// POUs/BACnet Objects/Local (Server)/Extended Process Data/FB_BACnet_PulseConverter_EX
FUNCTION_BLOCK FB_BACnet_PulseConverter_EX
VAR_IN_OUT
	Device				: FB_BACnet_Device;
END_VAR
VAR_OUTPUT
	bReady				: BOOL;
	fPresentValue		: REAL;
	bHighLimitEn		: BOOL;
	fHighLimit			: REAL;
	bLowLimitEn			: BOOL;
	fLowLimit			: REAL;
	fAdjustValue		: REAL;
	nCount				: UDINT;
	nCountBeforeChg		: UDINT;
	bOverridden			: BOOL;
	bOutOfService		: BOOL;
	bFault				: BOOL;
	bInAlarm			: BOOL;
	bOverRange			: BOOL;
	bUnderRange			: BOOL;
	bNoSensor			: BOOL;
	bOpenLoop			: BOOL;
	bShortedLoop		: BOOL;
	bCommFailure		: BOOL;
	bConfigError		: BOOL;
	bOtherFault			: BOOL;
	eEventState			: E_BACNETEVENTSTATE;
	bAckedTrans_ToOffNormal : BOOL;
	bAckedTrans_ToFault		: BOOL;
	bAckedTrans_ToNormal	: BOOL;
	tObjectID			: T_BACnet_ObjectIdentifier := 16#FFFFFFFF;
	bError				: BOOL;
	nErrorId			: UINT;
END_VAR
VAR
	_PresentValueIn AT%I*: REAL; 	(* ~(BACnet_PresentValue 		:		: )
								   		(BACnet_ObjectType 			: PC	: )	*)
	_HighLimit AT%I*: REAL;			(* ~(BACnet_HighLimit			:		: )	*)
	_LowLimit AT%I*: REAL;			(* ~(BACnet_LowLimit			:		: )	*)
	_AdjustValue AT%I*: REAL;		(* ~(BACnet_AdjustValue 		:		: ) *)
	_Count AT%I*: UDINT;			(* ~(BACnet_Count		 		:		: ) *)
	_CountBeforeChange AT%I*: UDINT;(* ~(BACnet_CountBeforeChange	:		: ) *)
	_ObjectId AT%I* : DWORD;		(* ~(BACnet_ObjectIdentifier	:		: LINK) *)
	_StatusFlags AT%I*: WORD; 		(* ~(BACnet_StatusFlags 		:		: )	*)
	_AckedTransitions AT%I*:WORD;	(* ~(BACnet_AckedTransitions	:		: ) *)
	_EventState AT%I*: WORD; 		(* ~(BACnet_EventState			:		: )	*)
	_LimitEnable AT%I*: WORD;		(* ~(BACnet_LimitEnable			:		: )	*)
	_Reliability AT%I*: WORD;;		(* ~(BACnet_Reliability 		:		: )	*)
	_AckedTransBits : ST_BACnet_EventTransitionBits;
	_StatusFlagsBits : ST_BACnet_StatusFlags;
	_LimitEnableBits : ST_BACnet_LimitEnable;
	_nUpdateCount : UDINT := 0;
END_VAR

(* update server device *)
IF (Device._nUpdateCount = _nUpdateCount) THEN
	Device();
END_IF
(* remind current number of update counter *)
_nUpdateCount := Device._nUpdateCount;

IF Device.bFirstCycle THEN
	(* first call of the server device since reboot/reset *)
	bReady := FALSE;

ELSIF (F_BACnet_GetObjType(_ObjectId) <> BACnetObjectType_PulseConverter) THEN
	(* wrong mapping / invalid object ID *)
	IF _ObjectId = 0 THEN
		nErrorId := BACnet_ERR_WRONG_MAPPING;
	ELSE
		nErrorId := BACnet_ERR_INVALID_OBJECTID;
	END_IF
	bReady := FALSE;
	tObjectID := 16#FFFFFFFF;

ELSIF (_StatusFlags < 4) THEN
	(* wrong mapping *)
	nErrorId := BACnet_ERR_WRONG_MAPPING;
	bReady := FALSE;

ELSIF Device.bOperational THEN
	(* ready state *)
	bReady := TRUE;
	nErrorId := BACnet_ERR_NO_ERROR;

	(* present value *)
	fPresentValue := _PresentValueIn;

	(* build bit states *)
	_StatusFlagsBits := F_BACnet_StatusFlags(_StatusFlags);
	_AckedTransBits := F_BACnet_EventTransitionFlags(_AckedTransitions);
	_LimitEnableBits :=	F_BACnet_LimitEnableFlags(_LimitEnable);

	(* copy states to output *)
	bHighLimitEn:= _LimitEnableBits.highLimitEnable;
	bLowLimitEn	:= _LimitEnableBits.lowLimitEnable;
	bOverridden	:= _StatusFlagsBits.overridden;
	bOutOfService:= _StatusFlagsBits.out_of_service;
	bFault		:= _StatusFlagsBits.fault;
	bInAlarm	:= _StatusFlagsBits.in_alarm;
	bOverRange	:= (_Reliability = TO_WORD(BACnetReliability_over_range));
	bUnderRange	:= (_Reliability = TO_WORD(BACnetReliability_under_range));
	bNoSensor	:= (_Reliability = TO_WORD(BACnetReliability_no_sensor));
	bOpenLoop	:= (_Reliability = TO_WORD(BACnetReliability_open_loop));
	bShortedLoop:= (_Reliability = TO_WORD(BACnetReliability_shorted_loop));
	bCommFailure := (_Reliability = TO_WORD(BACnetReliability_communication_failure));
	bConfigError:= (_Reliability = TO_WORD(BACnetReliability_configuration_error));
	bOtherFault	:= (_Reliability = TO_WORD(BACnetReliability_unreliable_other));
	bAckedTrans_ToOffNormal := _AckedTransBits.to_offnormal;
	bAckedTrans_ToFault := _AckedTransBits.to_fault;
	bAckedTrans_ToNormal := _AckedTransBits.to_normal;

	(* convert enumeration *)
	eEventState := TO_INT(_EventState);

	(* additional information *)
	fHighLimit			:= _HighLimit;
	fLowLimit			:= _LowLimit;
	fAdjustValue		:= _AdjustValue;
	nCount				:= _Count;
	nCountBeforeChg		:= _CountBeforeChange;
	tObjectID		:= F_BACnet_GetObjInstance(_ObjectId);

ELSE
	(* server device not ready, reset local ready flag *)
	bReady := FALSE;
	nErrorId := BACnet_ERR_OPERATIONAL;
END_IF
(* set error flag *)
bError := (nErrorId <> BACnet_ERR_NO_ERROR);

END_FUNCTION_BLOCK

// POUs/BACnet Objects/Local (Server)/Extended Process Data/FB_BACnet_Schedule_EX
FUNCTION_BLOCK FB_BACnet_Schedule_EX
VAR_IN_OUT
	Device				: FB_BACnet_Device;
END_VAR
VAR_OUTPUT
	bReady				: BOOL;
	bPresentValue		: BOOL;
	bOverridden			: BOOL;
	bOutOfService		: BOOL;
	bFault				: BOOL;
	bInAlarm			: BOOL;
	bConfigError		: BOOL;
	bOtherFault			: BOOL;
	tObjectID			: T_BACnet_ObjectIdentifier := 16#FFFFFFFF;
	bError				: BOOL;
	nErrorId			: UINT;
END_VAR
VAR
	_ObjectId AT%I*: DWORD;		(* ~(BACnet_ObjectIdentifier		:		: LINK) *)
	_Reliability AT%I*: WORD;; 	(* ~(BACnet_Reliability 			:		: )	*)
	_StatusFlags AT%I*: WORD; 	(* ~(BACnet_StatusFlags 			:		: )	*)
	_PresentValue AT%I*: BOOL;	(* ~(BACnet_PresentValueBool 		:		: )
									(BACnet_ObjectType 				: SCHED	: )	*)
	_StatusFlagsBits : ST_BACnet_StatusFlags;
	_nUpdateCount : UDINT := 0;
END_VAR

(* update server device *)
IF (Device._nUpdateCount = _nUpdateCount) THEN
	Device();
END_IF
(* remind current number of update counter *)
_nUpdateCount := Device._nUpdateCount;

(* check object type *)
IF (F_BACnet_GetObjType(_ObjectId) <> BACnetObjectType_Schedule) THEN
	(* wrong mapping / invalid object ID *)
	IF _ObjectId = 0 THEN
		nErrorId := BACnet_ERR_WRONG_MAPPING;
	ELSE
		nErrorId := BACnet_ERR_INVALID_OBJECTID;
	END_IF
	bReady := FALSE;

ELSIF (_StatusFlags < 4) THEN
	(* wrong mapping *)
	nErrorId := BACnet_ERR_WRONG_MAPPING;
	bReady := FALSE;

ELSIF Device.bOperational THEN
	(* ready state *)
	bReady := TRUE;
	nErrorId := BACnet_ERR_NO_ERROR;

	(* present value *)
	bPresentValue := _PresentValue;

	(* build bit states *)
	_StatusFlagsBits := F_BACnet_StatusFlags(_StatusFlags);

	(* copy states to output *)
	bOverridden := _StatusFlagsBits.overridden;
	bOutOfService := _StatusFlagsBits.out_of_service;
	bFault := _StatusFlagsBits.fault;
	bInAlarm := _StatusFlagsBits.in_alarm;
	bConfigError := (_Reliability = TO_WORD(BACnetReliability_configuration_error));
	bOtherFault := (_Reliability = TO_WORD(BACnetReliability_unreliable_other));
	tObjectID := _ObjectId;

ELSE
	bReady := FALSE;
	nErrorId := BACnet_ERR_OPERATIONAL;
END_IF
(* set error flag *)
bError := (nErrorId <> BACnet_ERR_NO_ERROR);

END_FUNCTION_BLOCK

// POUs/BACnet Objects/Local (Server)/Extended Process Data/FB_BACnet_TrendLog_EX
FUNCTION_BLOCK FB_BACnet_TrendLog_EX
VAR_IN_OUT
	Device	: FB_BACnet_Device;
END_VAR
VAR_OUTPUT
	bReady			: BOOL;
	bLogEnable		: BOOL;
	nRecordCount	: UDINT;
	nTotalCount		: UDINT;
	eEventState		: E_BACNETEVENTSTATE;
	bAckedTrans_ToOffNormal : BOOL;
	bAckedTrans_ToFault		: BOOL;
	bAckedTrans_ToNormal	: BOOL;
	tObjectID		: T_BACnet_ObjectIdentifier := 16#FFFFFFFF;
	bError			: BOOL;
	nErrorId		: UINT;
END_VAR
VAR
	_RecordCount AT%I*: UDINT;		(* ~(BACnet_RecordCount			:		: )
										(BACnet_ObjectType			: TLOG	: )	*)
	_TotalRecordCount AT%I*: UDINT;	(* ~(BACnet_TotalRecordCount	:		: )	*)
	_ObjectId AT%I*: DWORD;			(* ~(BACnet_ObjectIdentifier	:		: LINK) *)
	_EventState AT%I*: WORD;		(* ~(BACnet_EventState			:		: )	*)
	_AckedTransitions AT%I*:WORD;	(* ~(BACnet_AckedTransitions	:		: ) *)
	_LogEnable AT%I*: BOOL;			(* ~(BACnet_LogEnable			: 		: )	*)
	_AckedTransBits : ST_BACnet_EventTransitionBits;
	_nUpdateCount : UDINT := 0;
END_VAR

(* update server device *)
IF (Device._nUpdateCount = _nUpdateCount) THEN
	Device();
END_IF
(* remind current number of update counter *)
_nUpdateCount := Device._nUpdateCount;

(* check object type *)
IF (F_BACnet_GetObjType(_ObjectId) <> BACnetObjectType_TrendLog) THEN
	(* wrong mapping / invalid object ID *)
	IF _ObjectId = 0 THEN
		nErrorId := BACnet_ERR_WRONG_MAPPING;
	ELSE
		nErrorId := BACnet_ERR_INVALID_OBJECTID;
	END_IF
	bReady := FALSE;

ELSIF Device.bOperational THEN
	(* ready state *)
	bReady := TRUE;
	bLogEnable := _LogEnable;
	nErrorId := BACnet_ERR_NO_ERROR;

	(* build bit states *)
	_AckedTransBits		:= F_BACnet_EventTransitionFlags(_AckedTransitions);
	bAckedTrans_ToOffNormal := _AckedTransBits.to_offnormal;
	bAckedTrans_ToFault := _AckedTransBits.to_fault;
	bAckedTrans_ToNormal := _AckedTransBits.to_normal;
	tObjectID := _ObjectId;

	(* convert enumeration *)
	eEventState := TO_INT(_EventState);

	(* other states *)
	nRecordCount := _RecordCount;
	nTotalCount := _TotalRecordCount;

ELSE
	bReady := FALSE;
	nErrorId := BACnet_ERR_OPERATIONAL;
END_IF
(* set error flag *)
bError := (nErrorId <> BACnet_ERR_NO_ERROR);

END_FUNCTION_BLOCK

// POUs/BACnet Objects/Local (Server)/R6/FB_BACnet_Accumulator_R6
FUNCTION_BLOCK FB_BACnet_Accumulator_R6
VAR_INPUT
	nPV					: UDINT; (* number for present_value *)
END_VAR
VAR_IN_OUT
	Device				: FB_BACnet_Device;
END_VAR
VAR_OUTPUT
	bReady				: BOOL;
	nPresentValue		: UDINT;
	bOverridden			: BOOL;
	bOutOfService		: BOOL;
	bFault				: BOOL;
	bInAlarm			: BOOL;
	bError				: BOOL;
	nErrorId			: UINT;
END_VAR
VAR
	_PresentValueIn AT%I*:UDINT;	(* ~(BACnet_PresentValue	:		: )
										(BACnet_MaxPresValue	:		: writeprotect,nolink)
										(BACnet_ObjectType		: ACC	: )	*)
    _PresentValueOut AT%Q*:UDINT;	(* ~(BACnet_PresentValue	:		: )	*)
	_StatusFlags AT%I*:WORD;		(* ~(BACnet_StatusFlags		:		: )	*)
	_StatusFlagsBits : ST_BACnet_StatusFlags;

	_nUpdateCount : UDINT := 0;
END_VAR

(* update device *)
IF (Device._nUpdateCount = _nUpdateCount) THEN
	Device();
END_IF
(* remind current number of update counter *)
_nUpdateCount := Device._nUpdateCount;

IF _StatusFlags < 4 THEN
	(* mapping seems to be wrong (bit string for status flags must be 4 in minimum) *)
	nErrorId := BACnet_ERR_WRONG_MAPPING;

ELSIF Device.bOperational THEN
	(* clear error flag *)
	nErrorId := BACnet_ERR_NO_ERROR;
	bReady := TRUE;
	(* copy present value *)
	nPresentValue 		:= _PresentValueIn;
	_PresentValueOut	:= nPV;

	(* build bit states *)
	_StatusFlagsBits	:= F_BACnet_StatusFlags(_StatusFlags);

	(* copy states to output *)
	bOverridden := _StatusFlagsBits.overridden;
	bOutOfService := _StatusFlagsBits.out_of_service;
	bFault := _StatusFlagsBits.fault;
	bInAlarm := _StatusFlagsBits.in_alarm;
ELSE
	bReady := FALSE;
	(* and set error ID *)
	nErrorId := BACnet_ERR_OPERATIONAL;
END_IF

(* set error flag *)
bError := (nErrorId <> BACnet_ERR_NO_ERROR);

END_FUNCTION_BLOCK

// POUs/BACnet Objects/Local (Server)/R6/FB_BACnet_Accumulator_RAW_R6
FUNCTION_BLOCK FB_BACnet_Accumulator_RAW_R6
VAR_INPUT
	nPV					: UDINT; (* number for present_value *)
	nReliability		: WORD;
	bOutOfServiceOut	: BOOL;
END_VAR
VAR_IN_OUT
	Device				: FB_BACnet_Device;
END_VAR
VAR_OUTPUT
	bReady				: BOOL;
	nPresentValue		: UDINT;
	nMaxPV				: UDINT;
	bOverridden			: BOOL;
	bOutOfService		: BOOL;
	bFault				: BOOL;
	bInAlarm			: BOOL;
	bOverRange			: BOOL;
	bUnderRange			: BOOL;
	bNoSensor			: BOOL;
	bOpenLoop			: BOOL;
	bShortedLoop		: BOOL;
	bOtherFault			: BOOL;
	eEventState			: E_BACNETEVENTSTATE;
	bError				: BOOL;
	nErrorId			: UINT;
END_VAR
VAR
	_PresentValueIn AT%I*:UDINT;	(* ~(BACnet_PresentValue	:		: )
										(BACnet_ObjectType		: ACC	: )	*)
    _PresentValueOut AT%Q*:UDINT;	(* ~(BACnet_PresentValue	:		: )	*)
	_MaxPresValue AT%I*:UDINT;		(* ~(BACnet_MaxPresValue	:		: writeprotect) *)
	_StatusFlags AT%I*:WORD;		(* ~(BACnet_StatusFlags		:		: )	*)
	_EventState AT%I*: WORD; 		(* ~(BACnet_EventState 		:		: )	*)
	_Reliability AT%I*: WORD;; 		(* ~(BACnet_Reliability 	:		: )	*)
	_StatusFlagsOut AT%Q*:WORD;		(* ~(BACnet_StatusFlags		:		: )	*)
	_EventStateOut AT%Q*: WORD;		(* ~(BACnet_EventState 		:		: )	*)
	_ReliabilityOut AT%Q*: WORD;	(* ~(BACnet_Reliability 	:		: )	*)
	_OutOfServiceOut AT%Q*: BOOL;	(* ~(BACnet_OutOfService	:		: writeprotect) *)
	_StatusFlagsBits : ST_BACnet_StatusFlags;
	_StatusFlagsOutBits : ST_BACnet_StatusFlags;
	_nUpdateCount : UDINT := 0;
END_VAR

(* update client device *)
IF (Device._nUpdateCount = _nUpdateCount) THEN
	Device();
END_IF
(* remind current number of update counter *)
_nUpdateCount := Device._nUpdateCount;

(* copy reliability and out of service flags *)
_ReliabilityOut		:= nReliability;
_OutOfServiceOut	:= bOutOfServiceOut;

IF _StatusFlags < 4 THEN
	(* mapping seems to be wrong (bit string for status flags must be 4 in minimum) *)
	nErrorId := BACnet_ERR_WRONG_MAPPING;

ELSIF Device.bOperational THEN
	(* clear error flag *)
	nErrorId := BACnet_ERR_NO_ERROR;
	bReady := TRUE;
	(* copy present value *)
	nPresentValue 		:= _PresentValueIn;
	_PresentValueOut	:= nPV;
	nMaxPV				:= _MaxPresValue;

	(* build bit states *)
	_StatusFlagsBits	:= F_BACnet_StatusFlags(_StatusFlags);

	(* copy states to output *)
	bOverridden := _StatusFlagsBits.overridden;
	bOutOfService := _StatusFlagsBits.out_of_service;
	bFault := _StatusFlagsBits.fault;
	bInAlarm := _StatusFlagsBits.in_alarm;
	bOverRange := (_Reliability = TO_WORD(BACnetReliability_over_range));
	bUnderRange := (_Reliability = TO_WORD(BACnetReliability_under_range));
	bNoSensor := (_Reliability = TO_WORD(BACnetReliability_no_sensor));
	bOpenLoop := (_Reliability = TO_WORD(BACnetReliability_open_loop));
	bShortedLoop := (_Reliability = TO_WORD(BACnetReliability_shorted_loop));
	bOtherFault := (_Reliability = TO_WORD(BACnetReliability_unreliable_other));

	(* convert enumeration *)
	eEventState := TO_INT(_EventState);
ELSE
	bReady := FALSE;
	(* and set error ID *)
	nErrorId := BACnet_ERR_OPERATIONAL;
END_IF

(* set status flags depending on reliability *)
IF TO_INT(_ReliabilityOut) = BACnetReliability_no_fault_detected THEN
	_StatusFlagsOutBits.fault := FALSE;
	_StatusFlagsOutBits.in_alarm := FALSE;
	_EventStateOut := 0;
ELSE
	_StatusFlagsOutBits.fault := TRUE;
	_StatusFlagsOutBits.in_alarm := TRUE;
	_EventStateOut := 1;
END_IF

_StatusFlagsOutBits.out_of_service := _OutOfServiceOut;
_StatusFlagsOut	:= F_BACnet_GetStatusFlagsData(_StatusFlagsOutBits);

(* set error flag *)
bError := (nErrorId <> BACnet_ERR_NO_ERROR);

END_FUNCTION_BLOCK

// POUs/BACnet Objects/Local (Server)/RAW/FB_BACnet_Accumulator_RAW
FUNCTION_BLOCK FB_BACnet_Accumulator_RAW
VAR_INPUT
	nRawIn				AT%Q*: UINT; (* ~(BACnet_RawIoAccumulatorUnsignedValue : : ) *)
	bNoSensor			: BOOL;
	bOverRange			: BOOL;
	bUnderRange			: BOOL;
	bOpenLoop			: BOOL;
	bShortedLoop		: BOOL;
	bCommFailure		: BOOL;
	bOtherFault			: BOOL;
END_VAR
VAR_IN_OUT
	Device				: FB_BACnet_Device;
END_VAR
VAR_OUTPUT
	bReady				: BOOL;
	nPresentValue		: UDINT;
	bOverridden			: BOOL;
	bOutOfService		: BOOL;
	bFault				: BOOL;
	bInAlarm			: BOOL;
	bError				: BOOL;
	nErrorId			: UINT;
END_VAR
VAR
	_PresentValueIn AT%I*:UDINT;	(* ~(BACnet_PresentValue	:		: )
										(BACnet_MaxPresValue	:		: writeprotect,nolink)
										(BACnet_ObjectType		: ACC	: )	*)
	_ObjectId AT%I*: DWORD;			(* ~(BACnet_ObjectIdentifier:		: LINK) *)
	_StatusFlags AT%I*:WORD;		(* ~(BACnet_StatusFlags		:		: )	*)
	_ReliabilityIn AT%I*: WORD;		(* ~(BACnet_Reliability 	:		: )	*)
	_ReliabilityOut AT%Q*: WORD := INT_TO_WORD(BACnetReliability_no_fault_detected);(* ~(BACnet_Reliability 	:		: )	*)
	_StatusFlagsBits : ST_BACnet_StatusFlags;

	_nUpdateCount : UDINT := 0;
END_VAR

(* update device *)
IF Device._nUpdateCount = _nUpdateCount THEN
	Device();
END_IF
(* remind current number of update counter *)
_nUpdateCount := Device._nUpdateCount;

(* handle raw error *)
IF bNoSensor THEN
	_ReliabilityOut := TO_WORD(BACnetReliability_no_sensor);
ELSIF bOverRange THEN
	_ReliabilityOut := TO_WORD(BACnetReliability_over_range);
ELSIF bUnderRange THEN
	_ReliabilityOut := TO_WORD(BACnetReliability_under_range);
ELSIF bOpenLoop THEN
	_ReliabilityOut := TO_WORD(BACnetReliability_open_loop);
ELSIF bShortedLoop THEN
	_ReliabilityOut := TO_WORD(BACnetReliability_shorted_loop);
ELSIF bCommFailure THEN
	_ReliabilityOut := TO_WORD(BACnetReliability_communication_failure);
ELSIF bOtherFault THEN
	_ReliabilityOut := TO_WORD(BACnetReliability_unreliable_other);
ELSE
	_ReliabilityOut := TO_WORD(BACnetReliability_no_fault_detected);
END_IF

IF _StatusFlags < 4 THEN
	(* mapping seems to be wrong (bit string for status flags must be 4 in minimum) *)
	nErrorId := BACnet_ERR_WRONG_MAPPING;

ELSIF Device.bOperational THEN
	(* clear error flag *)
	nErrorId := BACnet_ERR_NO_ERROR;
	bReady := TRUE;
	(* copy present value *)
	nPresentValue 		:= _PresentValueIn;

	(* build bit states *)
	_StatusFlagsBits	:= F_BACnet_StatusFlags(_StatusFlags);

	(* copy states to output *)
	bOverridden := _StatusFlagsBits.overridden;
	bOutOfService := _StatusFlagsBits.out_of_service;
	bFault := _StatusFlagsBits.fault;
	bInAlarm := _StatusFlagsBits.in_alarm;
ELSE
	bReady := FALSE;
	(* and set error ID *)
	nErrorId := BACnet_ERR_OPERATIONAL;
END_IF

(* set error flag *)
bError := (nErrorId <> BACnet_ERR_NO_ERROR);

END_FUNCTION_BLOCK

// POUs/BACnet Objects/Local (Server)/RAW/FB_BACnet_AnalogInput_RAW
FUNCTION_BLOCK FB_BACnet_AnalogInput_RAW
VAR_INPUT
	nRawIn			AT%Q*: INT; (* ~(BACnet_RawIoAnalogSignedValue : : ) *)
	bNoSensor		: BOOL;
	bOverRange		: BOOL;
	bUnderRange		: BOOL;
	bOpenLoop		: BOOL;
	bShortedLoop	: BOOL;
	bCommFailure	: BOOL;
	bOtherFault		: BOOL;
END_VAR
VAR_IN_OUT
	Device	: FB_BACnet_Device;
END_VAR
VAR_OUTPUT
	bReady			: BOOL;
	fPresentValue	: REAL;
	bOverridden		: BOOL;
	bOutOfService	: BOOL;
	bFault			: BOOL;
	bInAlarm		: BOOL;
	bAckedTrans_ToOffNormal : BOOL;
	bAckedTrans_ToFault		: BOOL;
	bAckedTrans_ToNormal	: BOOL;
	bError			: BOOL;
	nErrorId		: UINT;
END_VAR
VAR
	_Reliability AT%Q*: WORD := INT_TO_WORD(BACnetReliability_no_fault_detected);(* ~(BACnet_Reliability 	:		: )	*)
	_PresentValue AT%I*: REAL; 		(* ~(BACnet_PresentValue 	:		: )
								   		(BACnet_ObjectType 		: AI	: )	*)
	_ObjectId AT%I*: DWORD;			(* ~(BACnet_ObjectIdentifier:		: LINK) *)
	_AckedTransitions AT%I*:WORD;	(* ~(BACnet_AckedTransitions:		: ) *)
	_StatusFlags AT%I*: WORD; 		(* ~(BACnet_StatusFlags 	:		: )	*)
	_AckedTransBits : ST_BACnet_EventTransitionBits;
	_StatusFlagsBits : ST_BACnet_StatusFlags;
	_nUpdateCount : UDINT := 0;
END_VAR

(* update server device *)
IF (Device._nUpdateCount = _nUpdateCount) THEN
	Device();
END_IF
(* remind current number of update counter *)
_nUpdateCount := Device._nUpdateCount;

(* handle raw error *)
IF bNoSensor THEN
	_Reliability := TO_WORD(BACnetReliability_no_sensor);
ELSIF bOverRange THEN
	_Reliability := TO_WORD(BACnetReliability_over_range);
ELSIF bUnderRange THEN
	_Reliability := TO_WORD(BACnetReliability_under_range);
ELSIF bOpenLoop THEN
	_Reliability := TO_WORD(BACnetReliability_open_loop);
ELSIF bShortedLoop THEN
	_Reliability := TO_WORD(BACnetReliability_shorted_loop);
ELSIF bCommFailure THEN
	_Reliability := TO_WORD(BACnetReliability_communication_failure);
ELSIF bOtherFault THEN
	_Reliability := TO_WORD(BACnetReliability_unreliable_other);
ELSE
	_Reliability := TO_WORD(BACnetReliability_no_fault_detected);
END_IF

(* check BitString format of StatusFlags --> if StatusFlags are less than 4, object isn't linked correctly *)
IF (_StatusFlags < 4) THEN
	(* wrong mapping *)
	nErrorId := BACnet_ERR_WRONG_MAPPING;
	bReady := FALSE;

ELSIF Device.bOperational THEN
	(* ready state *)
	bReady := TRUE;
	nErrorId := BACnet_ERR_NO_ERROR;

	(* present value *)
	fPresentValue := _PresentValue;

	(* build bit states *)
	_StatusFlagsBits := F_BACnet_StatusFlags(_StatusFlags);
	_AckedTransBits		:= F_BACnet_EventTransitionFlags(_AckedTransitions);

	(* copy states to output *)
	bOverridden := _StatusFlagsBits.overridden;
	bOutOfService := _StatusFlagsBits.out_of_service;
	bFault := _StatusFlagsBits.fault;
	bInAlarm := _StatusFlagsBits.in_alarm;
	bAckedTrans_ToOffNormal := _AckedTransBits.to_offnormal;
	bAckedTrans_ToFault := _AckedTransBits.to_fault;
	bAckedTrans_ToNormal := _AckedTransBits.to_normal;
ELSE
	(* server device not ready, reset local ready also *)
	bReady := FALSE;
	nErrorId := BACnet_ERR_OPERATIONAL;
END_IF
(* set error flag *)
bError := (nErrorId <> BACnet_ERR_NO_ERROR);

END_FUNCTION_BLOCK

// POUs/BACnet Objects/Local (Server)/RAW/FB_BACnet_AnalogOutput_RAW
FUNCTION_BLOCK FB_BACnet_AnalogOutput_RAW
VAR_INPUT
	bEnablePV		: BOOL; (* enable present value with priority x in priority array, FALSE = priority x disable *)
	bNullPV			: BOOL; (* clear priority entry *)
	fPV				: REAL; (* decimal number for priority x, when input bEnablePV is TRUE *)
	bRawOverridden	AT%Q*: BOOL; (* ~(BACnet_RawIoStateOverride	:		: ) *)
	bNoOutput		: BOOL;
	bOpenLoop		: BOOL;
	bShortedLoop	: BOOL;
	bCommFailure	: BOOL;
	bOtherFault		: BOOL;
END_VAR
VAR_IN_OUT
	Device	: FB_BACnet_Device;
END_VAR
VAR_OUTPUT
	bReady			: BOOL;
	fPresentValue	: REAL;
	bOverridden		: BOOL;
	bOutOfService	: BOOL;
	bFault			: BOOL;
	bInAlarm		: BOOL;
	bAckedTrans_ToOffNormal : BOOL;
	bAckedTrans_ToFault		: BOOL;
	bAckedTrans_ToNormal	: BOOL;
	bError			: BOOL;
	nErrorId		: UINT;
	nRawOut			AT%I*: INT;			(* ~(BACnet_RawIoAnalogSignedValue : : ) *)
END_VAR
VAR
	_PresentValue AT%I*: REAL; 			(* ~(BACnet_PresentValue 			:		: )
								   			(BACnet_ObjectType 				: AO	: )	*)
	_ObjectId AT%I*: DWORD;				(* ~(BACnet_ObjectIdentifier		:		: LINK) *)
	_AckedTransitions AT%I*:WORD;		(* ~(BACnet_AckedTransitions		:		: ) *)
	_StatusFlags AT%I*: WORD; 			(* ~(BACnet_StatusFlags 			:		: )	*)
    _PresentValue_Priority12 AT%Q*: DWORD;(* ~(BACnet_PresentValue_Priority12:		: )	*)
	_Reliability AT%Q*: WORD := INT_TO_WORD(BACnetReliability_no_fault_detected);(* ~(BACnet_Reliability 	:		: )	*)
	_AckedTransBits : ST_BACnet_EventTransitionBits;
	_StatusFlagsBits : ST_BACnet_StatusFlags;
	_nUpdateCount : UDINT := 0;
END_VAR

(* update server device *)
IF (Device._nUpdateCount = _nUpdateCount) THEN
	Device();
END_IF
(* remind current number of update counter *)
_nUpdateCount := Device._nUpdateCount;

(* handle raw error *)
IF bNoOutput THEN
	_Reliability := TO_WORD(BACnetReliability_no_output);
ELSIF bOpenLoop THEN
	_Reliability := TO_WORD(BACnetReliability_open_loop);
ELSIF bShortedLoop THEN
	_Reliability := TO_WORD(BACnetReliability_shorted_loop);
ELSIF bCommFailure THEN
	_Reliability := TO_WORD(BACnetReliability_communication_failure);
ELSIF bOtherFault THEN
	_Reliability := TO_WORD(BACnetReliability_unreliable_other);
ELSE
	_Reliability := TO_WORD(BACnetReliability_no_fault_detected);
END_IF

IF Device.bFirstCycle THEN
	(* first call of the server device since reboot/reset *)
	bReady := FALSE;
	_PresentValue_Priority12 := F_BACnet_RealNothing();

ELSIF (_StatusFlags < 4) THEN
	(* wrong mapping *)
	nErrorId := BACnet_ERR_WRONG_MAPPING;
	bReady := FALSE;

ELSIF Device.bOperational THEN
	(* ready state *)
	bReady := TRUE;
	nErrorId := BACnet_ERR_NO_ERROR;

	(* write into priority array *)
	_PresentValue_Priority12 := F_BACnet_RealPV(bEnablePV, bNullPV, fPV);

	(* present value *)
	fPresentValue := _PresentValue;

	(* build bit states *)
	_StatusFlagsBits := F_BACnet_StatusFlags(_StatusFlags);
	_AckedTransBits		:= F_BACnet_EventTransitionFlags(_AckedTransitions);

	(* copy states to output *)
	bOverridden := _StatusFlagsBits.overridden;
	bOutOfService := _StatusFlagsBits.out_of_service;
	bFault := _StatusFlagsBits.fault;
	bInAlarm := _StatusFlagsBits.in_alarm;
	bAckedTrans_ToOffNormal := _AckedTransBits.to_offnormal;
	bAckedTrans_ToFault := _AckedTransBits.to_fault;
	bAckedTrans_ToNormal := _AckedTransBits.to_normal;

ELSE
	(* server device not ready, reset local ready also *)
	bReady := FALSE;
	nErrorId := BACnet_ERR_OPERATIONAL;
END_IF
(* set error flag *)
bError := (nErrorId <> BACnet_ERR_NO_ERROR);

END_FUNCTION_BLOCK

// POUs/BACnet Objects/Local (Server)/RAW/FB_BACnet_BinaryInput_RAW
FUNCTION_BLOCK FB_BACnet_BinaryInput_RAW
VAR_INPUT
	bRawIn			AT%Q*: BOOL; (* ~(BACnet_RawIoBinaryBoolValue : : ) *)
	bNoSensor		: BOOL;
	bOpenLoop		: BOOL;
	bShortedLoop	: BOOL;
	bCommFailure	: BOOL;
	bOtherFault		: BOOL;
END_VAR
VAR_IN_OUT
	Device	: FB_BACnet_Device;
END_VAR
VAR_OUTPUT
	bReady			: BOOL;
	bPresentValue	: BOOL;
	bOverridden		: BOOL;
	bOutOfService	: BOOL;
	bFault			: BOOL;
	bInAlarm		: BOOL;
	bAckedTrans_ToOffNormal : BOOL;
	bAckedTrans_ToFault		: BOOL;
	bAckedTrans_ToNormal	: BOOL;
	bError			: BOOL;
	nErrorId		: UINT;
END_VAR
VAR
	_Reliability AT%Q*: WORD := INT_TO_WORD(BACnetReliability_no_fault_detected);(* ~(BACnet_Reliability 	:		: )	*)
	_ObjectId AT%I*: DWORD;				(* ~(BACnet_ObjectIdentifier	:		: LINK) *)
	_PresentValue AT%I*: WORD; 			(* ~(BACnet_PresentValue 		:		: )
											(BACnet_ObjectType			:BI    	: )	*)
	_StatusFlags AT%I*: WORD; 			(* ~(BACnet_StatusFlags 		:	    : )	*)
	_AckedTransitions AT%I*:WORD;		(* ~(BACnet_AckedTransitions	:		: ) *)
	_AckedTransBits : ST_BACnet_EventTransitionBits;
	_StatusFlagsBits : ST_BACnet_StatusFlags;
	_nUpdateCount : UDINT := 0;
END_VAR

(* update server device *)
IF (Device._nUpdateCount = _nUpdateCount) THEN
	Device();
END_IF
(* remind current number of update counter *)
_nUpdateCount := Device._nUpdateCount;

(* handle raw error *)
IF bNoSensor THEN
	_Reliability := TO_WORD(BACnetReliability_no_sensor);
ELSIF bOpenLoop THEN
	_Reliability := TO_WORD(BACnetReliability_open_loop);
ELSIF bShortedLoop THEN
	_Reliability := TO_WORD(BACnetReliability_shorted_loop);
ELSIF bCommFailure THEN
	_Reliability := TO_WORD(BACnetReliability_communication_failure);
ELSIF bOtherFault THEN
	_Reliability := TO_WORD(BACnetReliability_unreliable_other);
ELSE
	_Reliability := TO_WORD(BACnetReliability_no_fault_detected);
END_IF

(* check BitString format of StatusFlags --> if StatusFlags are less than 4, object isn't linked correctly *)
IF (_StatusFlags < 4) THEN
	(* wrong mapping *)
	nErrorId := BACnet_ERR_WRONG_MAPPING;
	bReady := FALSE;

ELSIF Device.bOperational THEN
	(* ready state *)
	bReady := TRUE;
	nErrorId := BACnet_ERR_NO_ERROR;

	(* present value *)
	bPresentValue := F_BinPV_To_Bool(TO_INT(_PresentValue));

	(* build bit states *)
	_StatusFlagsBits := F_BACnet_StatusFlags(_StatusFlags);
	_AckedTransBits		:= F_BACnet_EventTransitionFlags(_AckedTransitions);

	(* copy states to output *)
	bOverridden := _StatusFlagsBits.overridden;
	bOutOfService := _StatusFlagsBits.out_of_service;
	bFault := _StatusFlagsBits.fault;
	bInAlarm := _StatusFlagsBits.in_alarm;
	bAckedTrans_ToOffNormal := _AckedTransBits.to_offnormal;
	bAckedTrans_ToFault := _AckedTransBits.to_fault;
	bAckedTrans_ToNormal := _AckedTransBits.to_normal;

ELSE
	bReady := FALSE;
	nErrorId := BACnet_ERR_OPERATIONAL;
END_IF
(* set error flag *)
bError := (nErrorId <> BACnet_ERR_NO_ERROR);

END_FUNCTION_BLOCK

// POUs/BACnet Objects/Local (Server)/RAW/FB_BACnet_BinaryOutput_RAW
FUNCTION_BLOCK FB_BACnet_BinaryOutput_RAW
VAR_INPUT
	bEnablePV		: BOOL; (* enable present value with priority x in priority array, FALSE = priority x disable *)
	bNullPV			: BOOL; (* clear priority entry *)
	bPV				: BOOL; (* present value bool type *)
	bFeedback		AT%Q*:BOOL;	(* ~(BACnet_FeedbackValue : : ) *)
	bRawOverridden	AT%Q*: BOOL; (* ~(BACnet_RawIoStateOverride	:		: ) *)
	bNoOutput		: BOOL;
	bOpenLoop		: BOOL;
	bShortedLoop	: BOOL;
	bCommFailure	: BOOL;
	bOtherFault		: BOOL;
END_VAR
VAR_IN_OUT
	Device		: FB_BACnet_Device;
END_VAR
VAR_OUTPUT
	bReady			: BOOL;
	bPresentValue	: BOOL;
	bOverridden		: BOOL;
	bOutOfService	: BOOL;
	bFault			: BOOL;
	bInAlarm		: BOOL;
	bAckedTrans_ToOffNormal : BOOL;
	bAckedTrans_ToFault		: BOOL;
	bAckedTrans_ToNormal	: BOOL;
	bError			: BOOL;
	nErrorId		: UINT;
	bRawOut			AT%I*: BOOL;			(* ~(BACnet_RawIoBinaryBoolValue	:		: ) *)
END_VAR
VAR
	_ObjectId AT%I*: DWORD;					(* ~(BACnet_ObjectIdentifier		:		: LINK) *)
	_PresentValue AT%I*: WORD; 				(* ~(BACnet_PresentValue 			:		: )
								   				(BACnet_ObjectType 				: BO	: )	*)
	_StatusFlags AT%I*: WORD; 				(* ~(BACnet_StatusFlags 			:		: )	*)
	_AckedTransitions AT%I*:WORD;			(* ~(BACnet_AckedTransitions		:		: ) *)
    _PresentValue_Priority12 AT%Q*: WORD;	(* ~(BACnet_PresentValue_Priority12	:		: )	*)
	_Reliability AT%Q*: WORD := INT_TO_WORD(BACnetReliability_no_fault_detected);(* ~(BACnet_Reliability 	:		: )	*)
	_AckedTransBits : ST_BACnet_EventTransitionBits;
	_StatusFlagsBits : ST_BACnet_StatusFlags;
	_nUpdateCount : UDINT := 0;
END_VAR

(* update server device *)
IF (Device._nUpdateCount = _nUpdateCount) THEN
	Device();
END_IF
(* remind current number of update counter *)
_nUpdateCount := Device._nUpdateCount;

(* handle raw error *)
IF bNoOutput THEN
	_Reliability := TO_WORD(BACnetReliability_no_output);
ELSIF bOpenLoop THEN
	_Reliability := TO_WORD(BACnetReliability_open_loop);
ELSIF bShortedLoop THEN
	_Reliability := TO_WORD(BACnetReliability_shorted_loop);
ELSIF bCommFailure THEN
	_Reliability := TO_WORD(BACnetReliability_communication_failure);
ELSIF bOtherFault THEN
	_Reliability := TO_WORD(BACnetReliability_unreliable_other);
ELSE
	_Reliability := TO_WORD(BACnetReliability_no_fault_detected);
END_IF

IF Device.bFirstCycle THEN
	(* first call of the server device since reboot/reset *)
	bReady := FALSE;
	_PresentValue_Priority12 := to_word(BACnetBinaryPV_Nothing);

ELSIF (_StatusFlags < 4) THEN
	(* wrong mapping *)
	nErrorId := BACnet_ERR_WRONG_MAPPING;
	bReady := FALSE;

ELSIF Device.bOperational THEN
	(* ready state *)
	bReady := TRUE;
	nErrorId := BACnet_ERR_NO_ERROR;

	(* write into priority array *)
	_PresentValue_Priority12 := to_word(F_Bool_To_BinPV(bEnablePV, bNullPV, bPV));

	(* present value *)
	bPresentValue := F_BinPV_To_Bool(TO_INT(_PresentValue));

	(* build bit states *)
	_StatusFlagsBits := F_BACnet_StatusFlags(_StatusFlags);
	_AckedTransBits		:= F_BACnet_EventTransitionFlags(_AckedTransitions);

	(* copy states to output *)
	bOverridden := _StatusFlagsBits.overridden;
	bOutOfService := _StatusFlagsBits.out_of_service;
	bFault := _StatusFlagsBits.fault;
	bInAlarm := _StatusFlagsBits.in_alarm;
	bAckedTrans_ToOffNormal := _AckedTransBits.to_offnormal;
	bAckedTrans_ToFault := _AckedTransBits.to_fault;
	bAckedTrans_ToNormal := _AckedTransBits.to_normal;

ELSE
	(* server device not ready, reset local ready also *)
	bReady := FALSE;
	nErrorId := BACnet_ERR_OPERATIONAL;
END_IF
(* set error flag *)
bError := (nErrorId <> BACnet_ERR_NO_ERROR);

END_FUNCTION_BLOCK

// POUs/BACnet Objects/Local (Server)/RAW/FB_BACnet_MultiStateInput_RAW
FUNCTION_BLOCK FB_BACnet_MultiStateInput_RAW
VAR_INPUT
	nRawIn				AT%Q*: DWORD; (* ~(BACnet_PresentValue : : ) *)
	bNoSensor		: BOOL;
	bOverRange		: BOOL;
	bUnderRange		: BOOL;
	bOpenLoop		: BOOL;
	bShortedLoop	: BOOL;
	bCommFailure	: BOOL;
	bOtherFault		: BOOL;
END_VAR
VAR_IN_OUT
	Device				: FB_BACnet_Device;
END_VAR
VAR_OUTPUT
	bReady				: BOOL;
	nPresentValue		: UDINT;
	bOverridden			: BOOL;
	bOutOfService		: BOOL;
	bFault				: BOOL;
	bInAlarm			: BOOL;
	bAckedTrans_ToOffNormal : BOOL;
	bAckedTrans_ToFault		: BOOL;
	bAckedTrans_ToNormal	: BOOL;
	nNbrOfStates		: UDINT;
	bError				: BOOL;
	nErrorId			: UINT;
END_VAR
VAR
	_Reliability AT%Q*: WORD := INT_TO_WORD(BACnetReliability_no_fault_detected);(* ~(BACnet_Reliability 	:		: )	*)
	_PresentValue AT%I*: UDINT; 		(* ~(BACnet_PresentValue 	:		: )
								   			(BACnet_ObjectType 		: MI	: )	*)
	_NumberOfStates AT%I*: UDINT;		(* ~(BACnet_NumberOfStates	:		: )	*)
	_ObjectId AT%I*: DWORD;				(* ~(BACnet_ObjectIdentifier:		: LINK) *)
	_StatusFlags AT%I*: WORD; 			(* ~(BACnet_StatusFlags 	:		: )	*)
	_AckedTransitions AT%I*:WORD;		(* ~(BACnet_AckedTransitions:		: ) *)
	_AckedTransBits : ST_BACnet_EventTransitionBits;
	_nUpdateCount : UDINT := 0;
	_StatusFlagsBits : ST_BACnet_StatusFlags;
END_VAR

(* update server device *)
IF (Device._nUpdateCount = _nUpdateCount) THEN
	Device();
END_IF
(* remind current number of update counter *)
_nUpdateCount := Device._nUpdateCount;

(* handle raw error *)
IF bNoSensor THEN
	_Reliability := TO_WORD(BACnetReliability_no_sensor);
ELSIF bOverRange THEN
	_Reliability := TO_WORD(BACnetReliability_over_range);
ELSIF bUnderRange THEN
	_Reliability := TO_WORD(BACnetReliability_under_range);
ELSIF bOpenLoop THEN
	_Reliability := TO_WORD(BACnetReliability_open_loop);
ELSIF bShortedLoop THEN
	_Reliability := TO_WORD(BACnetReliability_shorted_loop);
ELSIF bCommFailure THEN
	_Reliability := TO_WORD(BACnetReliability_communication_failure);
ELSIF bOtherFault THEN
	_Reliability := TO_WORD(BACnetReliability_unreliable_other);
ELSE
	_Reliability := TO_WORD(BACnetReliability_no_fault_detected);
END_IF

(* check object type *)
IF (F_BACnet_GetObjType(_ObjectId) <> BACnetObjectType_MultiStateInput) THEN
	(* wrong mapping / invalid object ID *)
	IF _ObjectId = 0 THEN
		nErrorId := BACnet_ERR_WRONG_MAPPING;
	ELSE
		nErrorId := BACnet_ERR_INVALID_OBJECTID;
	END_IF
	bReady := FALSE;

ELSIF (_StatusFlags < 4) THEN
	(* wrong mapping *)
	nErrorId := BACnet_ERR_WRONG_MAPPING;
	bReady := FALSE;

ELSIF Device.bOperational THEN
	(* ready state *)
	bReady := TRUE;
	nErrorId := BACnet_ERR_NO_ERROR;

	(* present value *)
	nPresentValue := _PresentValue;

	(* build bit states *)
	_StatusFlagsBits := F_BACnet_StatusFlags(_StatusFlags);
	_AckedTransBits		:= F_BACnet_EventTransitionFlags(_AckedTransitions);

	(* copy states to output *)
	bOverridden := _StatusFlagsBits.overridden;
	bOutOfService := _StatusFlagsBits.out_of_service;
	bFault := _StatusFlagsBits.fault;
	bInAlarm := _StatusFlagsBits.in_alarm;
	bAckedTrans_ToOffNormal := _AckedTransBits.to_offnormal;
	bAckedTrans_ToFault := _AckedTransBits.to_fault;
	bAckedTrans_ToNormal := _AckedTransBits.to_normal;

	(* number of states *)
	nNbrOfStates := _NumberOfStates;

ELSE
	(* server device not ready, reset local ready also *)
	bReady := FALSE;
	nErrorId := BACnet_ERR_OPERATIONAL;
END_IF
(* set error flag *)
bError := (nErrorId <> BACnet_ERR_NO_ERROR);

END_FUNCTION_BLOCK

// POUs/BACnet Objects/Local (Server)/RAW/FB_BACnet_MultiStateOutput_RAW
FUNCTION_BLOCK FB_BACnet_MultiStateOutput_RAW
VAR_INPUT
	bEnablePV			: BOOL; (* enable present value with priority x in priority array, FALSE = priority x disable *)
	bNullPV				: BOOL; (* clear priority entry *)
	nPV					: UDINT; (* number for priority x, when input bEnablePV is TRUE *)
	nFeedback			AT%Q*: DWORD; (* ~(BACnet_FeedbackValue : : ) *)
	bNoOutput			: BOOL;
	bOpenLoop			: BOOL;
	bShortedLoop		: BOOL;
	bCommFailure		: BOOL;
	bOtherFault			: BOOL;
END_VAR
VAR_IN_OUT
	Device				: FB_BACnet_Device;
END_VAR
VAR_OUTPUT
	bReady				: BOOL;
	nPresentValue		: UDINT;
	bOverridden			: BOOL;
	bOutOfService		: BOOL;
	bFault				: BOOL;
	bInAlarm			: BOOL;
	bAckedTrans_ToOffNormal : BOOL;
	bAckedTrans_ToFault		: BOOL;
	bAckedTrans_ToNormal	: BOOL;
	nNbrOfStates		: UDINT;
	bError				: BOOL;
	nErrorId			: UINT;
	nRawOut				AT%I*: DWORD;		(* ~(BACnet_PresentValue		:		: ) *)
END_VAR
VAR
    _PresentValue_Priority12 AT%Q*: UDINT;	(* ~(BACnet_PresentValue_Priority12:	: )
								   				(BACnet_ObjectType			: MO	: )	*)
	_Reliability AT%Q*: WORD := INT_TO_WORD(BACnetReliability_no_fault_detected);(* ~(BACnet_Reliability 	:		: )	*)
	_NumberOfStates AT%I*: UDINT;			(* ~(BACnet_NumberOfStates		:		: )	*)
	_ObjectId AT%I*: DWORD;					(* ~(BACnet_ObjectIdentifier	:		: LINK) *)
	_StatusFlags AT%I*: WORD; 				(* ~(BACnet_StatusFlags			:		: )	*)
	_AckedTransitions AT%I*:WORD;			(* ~(BACnet_AckedTransitions	:		: ) *)
	_AckedTransBits : ST_BACnet_EventTransitionBits;
	_nUpdateCount : UDINT := 0;
	_StatusFlagsBits : ST_BACnet_StatusFlags;
END_VAR

(* update server device *)
IF (Device._nUpdateCount = _nUpdateCount) THEN
	Device();
END_IF
(* remind current number of update counter *)
_nUpdateCount := Device._nUpdateCount;

(* handle raw error *)
IF bNoOutput THEN
	_Reliability := TO_WORD(BACnetReliability_no_output);
ELSIF bOpenLoop THEN
	_Reliability := TO_WORD(BACnetReliability_open_loop);
ELSIF bShortedLoop THEN
	_Reliability := TO_WORD(BACnetReliability_shorted_loop);
ELSIF bCommFailure THEN
	_Reliability := TO_WORD(BACnetReliability_communication_failure);
ELSIF bOtherFault THEN
	_Reliability := TO_WORD(BACnetReliability_unreliable_other);
ELSE
	_Reliability := TO_WORD(BACnetReliability_no_fault_detected);
END_IF

(* check object type *)
IF Device.bFirstCycle THEN
	(* first call of the server device since reboot/reset *)
	bReady := FALSE;
	_PresentValue_Priority12 := 16#FFFFFFFF;

ELSIF (F_BACnet_GetObjType(_ObjectId) <> BACnetObjectType_MultiStateOutput) THEN
	(* wrong mapping / invalid object ID *)
	IF _ObjectId = 0 THEN
		nErrorId := BACnet_ERR_WRONG_MAPPING;
	ELSE
		nErrorId := BACnet_ERR_INVALID_OBJECTID;
	END_IF
	bReady := FALSE;

ELSIF (_StatusFlags < 4) THEN
	(* wrong mapping *)
	nErrorId := BACnet_ERR_WRONG_MAPPING;
	bReady := FALSE;

ELSIF Device.bOperational THEN
	(* ready state *)
	bReady := TRUE;
	nErrorId := BACnet_ERR_NO_ERROR;

	(* write into priority array *)
	_PresentValue_Priority12 := F_BACnet_MultiStatePV(bEnablePV, bNullPV, nPV);

	(* present value *)
	nPresentValue := nRawOut;

	(* build bit states *)
	_StatusFlagsBits := F_BACnet_StatusFlags(_StatusFlags);
	_AckedTransBits		:= F_BACnet_EventTransitionFlags(_AckedTransitions);

	(* copy states to output *)
	bOverridden := _StatusFlagsBits.overridden;
	bOutOfService := _StatusFlagsBits.out_of_service;
	bFault := _StatusFlagsBits.fault;
	bInAlarm := _StatusFlagsBits.in_alarm;
	bAckedTrans_ToOffNormal := _AckedTransBits.to_offnormal;
	bAckedTrans_ToFault := _AckedTransBits.to_fault;
	bAckedTrans_ToNormal := _AckedTransBits.to_normal;

	(* number of states *)
	nNbrOfStates := _NumberOfStates;

ELSE
	(* server device not ready, reset local ready also *)
	bReady := FALSE;
	nErrorId := BACnet_ERR_OPERATIONAL;
END_IF
(* set error flag *)
bError := (nErrorId <> BACnet_ERR_NO_ERROR);

END_FUNCTION_BLOCK

// POUs/BACnet Objects/Local (Server)/RAW/FB_BACnet_PulseConverter_RAW
FUNCTION_BLOCK FB_BACnet_PulseConverter_RAW
VAR_INPUT
	nRawIn			AT%Q*: UINT; (* ~(BACnet_RawIoPulseConverterUnsignedValue : : ) *)
	bNoSensor		: BOOL;
	bOverRange		: BOOL;
	bUnderRange		: BOOL;
	bOpenLoop		: BOOL;
	bShortedLoop	: BOOL;
	bCommFailure	: BOOL;
	bConfigError	: BOOL;
	bOtherFault		: BOOL;
END_VAR
VAR_IN_OUT
	Device			: FB_BACnet_Device;
END_VAR
VAR_OUTPUT
	bReady			: BOOL;
	fPresentValue	: REAL;
	nCount			: UDINT;
	bOverridden		: BOOL;
	bOutOfService	: BOOL;
	bFault			: BOOL;
	bInAlarm		: BOOL;
	bError			: BOOL;
	nErrorId		: UINT;
END_VAR
VAR
	_PresentValueIn AT%I*: REAL; 	(* ~(BACnet_PresentValue 		:		: )
								   		(BACnet_ObjectType 			: PC	: )
										(BACnet_InputReference		: 		: nolink, disable) *)
	_Count AT%I*: UDINT;			(* ~(BACnet_Count		 		:		: ) *)
	_ObjectId AT%I*: DWORD;			(* ~(BACnet_ObjectIdentifier	:		: LINK) *)
	_StatusFlags AT%I*: WORD; 		(* ~(BACnet_StatusFlags 		:		: )	*)
	_ReliabilityIn AT%I*: WORD;		(* ~(BACnet_Reliability 		:		: )	*)
	_ReliabilityOut AT%Q*: WORD := INT_TO_WORD(BACnetReliability_no_fault_detected);(* ~(BACnet_Reliability 	:		: )	*)
	_StatusFlagsBits : ST_BACnet_StatusFlags;
	_nUpdateCount : UDINT := 0;
END_VAR

(* update server device *)
IF (Device._nUpdateCount = _nUpdateCount) THEN
	Device();
END_IF
(* remind current number of update counter *)
_nUpdateCount := Device._nUpdateCount;

(* handle raw error *)
IF (_ReliabilityIn <> TO_WORD(BACnetReliability_configuration_error)) THEN
	IF bNoSensor THEN
		_ReliabilityOut := TO_WORD(BACnetReliability_no_sensor);
	ELSIF bOverRange THEN
		_ReliabilityOut := to_word(BACnetReliability_over_range);
	ELSIF bUnderRange THEN
		_ReliabilityOut := to_word(BACnetReliability_under_range);
	ELSIF bOpenLoop THEN
		_ReliabilityOut := to_word(BACnetReliability_open_loop);
	ELSIF bShortedLoop THEN
		_ReliabilityOut := to_word(BACnetReliability_shorted_loop);
	ELSIF bCommFailure THEN
		_ReliabilityOut := to_word(BACnetReliability_communication_failure);
	ELSIF bOtherFault THEN
		_ReliabilityOut := to_word(BACnetReliability_unreliable_other);
	ELSE
		_ReliabilityOut := to_word(BACnetReliability_no_fault_detected);
	END_IF
ELSE
	_ReliabilityOut := to_word(BACnetReliability_no_fault_detected);
END_IF

IF Device.bFirstCycle THEN
	(* first call of the server device since reboot/reset *)
	bReady := FALSE;

ELSIF (_StatusFlags < 4) THEN
	(* wrong mapping *)
	nErrorId := BACnet_ERR_WRONG_MAPPING;
	bReady := FALSE;

ELSIF Device.bOperational THEN
	(* ready state *)
	bReady := TRUE;
	nErrorId := BACnet_ERR_NO_ERROR;

	(* present value *)
	fPresentValue := _PresentValueIn;

	(* build bit states *)
	_StatusFlagsBits := F_BACnet_StatusFlags(_StatusFlags);

	(* copy states to output *)
	bOverridden		:= _StatusFlagsBits.overridden;
	bOutOfService	:= _StatusFlagsBits.out_of_service;
	bFault			:= _StatusFlagsBits.fault;
	bInAlarm		:= _StatusFlagsBits.in_alarm;

	(* additional information *)
	nCount			:= _Count;

ELSE
	(* server device not ready, reset local ready flag *)
	bReady := FALSE;
	nErrorId := BACnet_ERR_OPERATIONAL;
END_IF
(* set error flag *)
bError := (nErrorId <> BACnet_ERR_NO_ERROR);

END_FUNCTION_BLOCK

// POUs/BACnet Objects/Local (Server)/FB_BACnet_Accumulator
FUNCTION_BLOCK FB_BACnet_Accumulator EXTENDS _FB_BACnet_Object
VAR_INPUT
	nValueSet			: UDINT; (* number for present_value *)
END_VAR
VAR_OUTPUT
	nPresentValue		: UDINT;
END_VAR
VAR
	_PresentValueIn AT%I*:UDINT;	(* ~(BACnet_PresentValue	:		: )
										(BACnet_MaxPresValue	:		: writeprotect,nolink)
										(BACnet_ObjectType		: ACC	: )	*)
	_ValueSet AT%Q*:UDINT;			(* ~(BACnet_ValueSet		:		: ) *)
END_VAR

SUPER^(Device:=Device);
IF bReady THEN
	(* copy present value *)
	nPresentValue 		:= _PresentValueIn;
	_ValueSet			:= nValueSet;
END_IF

END_FUNCTION_BLOCK

// POUs/BACnet Objects/Local (Server)/FB_BACnet_AnalogInput
FUNCTION_BLOCK FB_BACnet_AnalogInput EXTENDS _FB_BACnet_AnalogObject
VAR
	_PresentValue AT%I*: REAL; 	(* ~(BACnet_ObjectType 		: AI	: )
									(BACnet_PresentValue 	:		: ) *)
END_VAR

SUPER^(Device:=Device);
IF bReady THEN
	fPresentValue := _PresentValue;
END_IF

END_FUNCTION_BLOCK

// POUs/BACnet Objects/Local (Server)/FB_BACnet_AnalogOutput
FUNCTION_BLOCK FB_BACnet_AnalogOutput EXTENDS _FB_BACnet_AnalogObject
VAR_INPUT
	bEnablePV		: BOOL; (* enable present value with priority x in priority array, FALSE = priority x disable *)
	bNullPV			: BOOL; (* clear priority entry *)
	fPV				: REAL; (* decimal number for priority x, when input bEnablePV is TRUE *)
END_VAR
VAR
	_PresentValue AT%I*: REAL; 			(* ~(BACnet_PresentValue 			:		: )
								   			(BACnet_ObjectType 				: AO	: )	*)
    _PresentValue_Priority12 AT%Q*: DWORD;(* ~(BACnet_PresentValue_Priority12:		: )	*)
END_VAR

SUPER^(Device := Device);
IF Device.bFirstCycle THEN
	(* first call of the server device since reboot/reset *)
	bReady := FALSE;
	_PresentValue_Priority12 := F_BACnet_RealNothing();

ELSIF bReady THEN
	(* write into priority array *)
	_PresentValue_Priority12 := F_BACnet_RealPV(bEnablePV, bNullPV, fPV);
	(* present value *)
	fPresentValue := _PresentValue;
END_IF

END_FUNCTION_BLOCK

// POUs/BACnet Objects/Local (Server)/FB_BACnet_AnalogValue
FUNCTION_BLOCK FB_BACnet_AnalogValue EXTENDS _FB_BACnet_AnalogObject
VAR_INPUT
	bEnablePV		: BOOL; (* enable present value with priority x in priority array, FALSE = priority x disable *)
	bNullPV			: BOOL; (* clear priority entry *)
	fPV				: REAL; (* decimal number for priority x, when input bEnablePV is TRUE *)
END_VAR
VAR
	_PresentValue AT%I*: REAL; 			(* ~(BACnet_PresentValue 			:		: )
								   			(BACnet_ObjectType 				: AV	: )	*)
    _PresentValue_Priority12 AT%Q*: DWORD;(* ~(BACnet_PresentValue_Priority12:		: )	*)
END_VAR

SUPER^(Device := Device);
IF Device.bFirstCycle THEN
	(* first call of the server device since reboot/reset *)
	bReady := FALSE;
	_PresentValue_Priority12 := F_BACnet_RealNothing();

ELSIF bReady THEN
	(* write into priority array *)
	_PresentValue_Priority12 := F_BACnet_RealPV(bEnablePV, bNullPV, fPV);
	(* present value *)
	fPresentValue := _PresentValue;
END_IF

END_FUNCTION_BLOCK

// POUs/BACnet Objects/Local (Server)/FB_BACnet_Averaging
FUNCTION_BLOCK FB_BACnet_Averaging
VAR_IN_OUT
	Device			: FB_BACnet_Device;
END_VAR
VAR_OUTPUT
	bReady			: BOOL;
	fAverageValue	: REAL;
	fMaximumValue	: REAL;
	fMinimumValue	: REAL;
	nValidSamples	: UDINT;
	nWindowSamples	: UDINT;
	nWindowInterval	: UDINT; (* [s] *)
	bError			: BOOL;
	nErrorId		: UINT;
END_VAR
VAR
	_AverageValue AT%I*: REAL;			(* ~(BACnet_AverageValue	:		: )
											(BACnet_ObjectType 		: AVG	: ) *)
	_MaximumValue AT%I*: REAL;			(* ~(BACnet_MaximumValue	:		: ) *)
	_MinimumValue AT%I*: REAL;			(* ~(BACnet_MinimumValue	:		: ) *)
	_ValidSamples AT%I*: UDINT;			(* ~(BACnet_ValidSamples	:		: ) *)
	_WindowSamples AT%I*: UDINT;		(* ~(BACnet_WindowSamples	:		: ) *)
	_WindowInterval AT%I*: UDINT;		(* ~(BACnet_WindowInterval	:		: ) *)
	_nUpdateCount : UDINT := 0;
END_VAR

(* update server device *)
IF (Device._nUpdateCount = _nUpdateCount) THEN
	Device();
END_IF
(* remind current number of update counter *)
_nUpdateCount := Device._nUpdateCount;

IF Device.bFirstCycle THEN
	(* first call of the server device since reboot/reset *)
	bReady := FALSE;
ELSIF Device.bOperational THEN
	(* ready state *)
	bReady := TRUE;
	nErrorId := BACnet_ERR_NO_ERROR;

	(* present values *)
	fAverageValue	:= _AverageValue;
	fMaximumValue	:= _MaximumValue;
	fMinimumValue	:= _MinimumValue;
	nValidSamples	:= _ValidSamples;
	nWindowSamples	:= _WindowSamples;
	nWindowInterval	:= _WindowInterval;

ELSE
	(* server device not ready, reset local ready also *)
	bReady := FALSE;
	nErrorId := BACnet_ERR_OPERATIONAL;
END_IF
(* set error flag *)
bError := (nErrorId <> BACnet_ERR_NO_ERROR);

END_FUNCTION_BLOCK

// POUs/BACnet Objects/Local (Server)/FB_BACnet_BinaryInput
FUNCTION_BLOCK FB_BACnet_BinaryInput EXTENDS _FB_BACnet_BinaryObject
VAR
	_PresentValue AT%I*: WORD; 			(* ~(BACnet_PresentValue 		:		: )
											(BACnet_ObjectType			: BI   	: )	*)
END_VAR

SUPER^(Device := Device);
IF bReady THEN
	(* present value *)
	bPresentValue := F_BinPV_To_Bool(TO_INT(_PresentValue));
END_IF

END_FUNCTION_BLOCK

// POUs/BACnet Objects/Local (Server)/FB_BACnet_BinaryOutput
FUNCTION_BLOCK FB_BACnet_BinaryOutput EXTENDS _FB_BACnet_BinaryObject
VAR_INPUT 
	bEnablePV		: BOOL; (* enable present value with priority x in priority array, FALSE = priority x disable *)
	bNullPV			: BOOL; (* clear priority entry *)
	bPV				: BOOL; (* present value bool type *)
END_VAR
VAR
	_PresentValue AT%I*: WORD; 			(* ~(BACnet_PresentValue 			:		: )
								   			(BACnet_ObjectType 				: BO	: )	*)
    _PresentValue_Priority12 AT%Q*: WORD;(* ~(BACnet_PresentValue_Priority12:		: )	*)
END_VAR

SUPER^(Device := Device);
IF Device.bFirstCycle THEN
	(* first call of the server device since reboot/reset *)
	bReady := FALSE;
	_PresentValue_Priority12 := INT_TO_WORD(BACnetBinaryPV_Nothing);

ELSIF bReady THEN
	(* write into priority array *)
	_PresentValue_Priority12 := INT_TO_WORD(F_Bool_To_BinPV(bEnablePV, bNullPV, bPV));

	(* present value *)
	bPresentValue := F_BinPV_To_Bool(TO_INT(_PresentValue));
END_IF

END_FUNCTION_BLOCK

// POUs/BACnet Objects/Local (Server)/FB_BACnet_BinaryValue
FUNCTION_BLOCK FB_BACnet_BinaryValue EXTENDS _FB_BACnet_BinaryObject
VAR_INPUT
	bEnablePV		: BOOL; (* enable present value with priority x in priority array, FALSE = priority x disable *)
	bNullPV			: BOOL; (* clear priority entry *)
	bPV				: BOOL; (* present value bool type *)
END_VAR
VAR
	_PresentValue AT%I*: WORD; 			(* ~(BACnet_PresentValue 			:		: )
								   			(BACnet_ObjectType 				: BV	: )	*)
    _PresentValue_Priority12 AT%Q*: WORD;(* ~(BACnet_PresentValue_Priority12:		: )	*)
END_VAR

SUPER^(Device := Device);
IF Device.bFirstCycle THEN
	(* first call of the server device since reboot/reset *)
	bReady := FALSE;
	_PresentValue_Priority12 := INT_TO_WORD(BACnetBinaryPV_Nothing);

ELSIF bReady THEN
	(* write into priority array *)
	_PresentValue_Priority12 := INT_TO_WORD(F_Bool_To_BinPV(bEnablePV, bNullPV, bPV));

	(* present value *)
	bPresentValue := F_BinPV_To_Bool(TO_INT(_PresentValue));
END_IF

END_FUNCTION_BLOCK

// POUs/BACnet Objects/Local (Server)/FB_BACnet_Calendar
FUNCTION_BLOCK FB_BACnet_Calendar
VAR_IN_OUT
	Device	: FB_BACnet_Device;
END_VAR
VAR_OUTPUT
	bReady			: BOOL;
	bPresentValue	: BOOL;
	bError			: BOOL;
	nErrorId		: UINT;
END_VAR
VAR
	_PresentValue AT%I*: BOOL;	(* ~(BACnet_PresentValue 			:		: )
									(BACnet_ObjectType 				: CAL	: )	*)
	_nUpdateCount : UDINT := 0;
END_VAR

(* update server device *)
IF (Device._nUpdateCount = _nUpdateCount) THEN
	Device();
END_IF
(* remind current number of update counter *)
_nUpdateCount := Device._nUpdateCount;

IF Device.bOperational THEN
	(* ready state *)
	bReady := TRUE;
	nErrorId := BACnet_ERR_NO_ERROR;
	(* present value *)
	bPresentValue := _PresentValue;
ELSE
	(* server device not ready, reset local ready also *)
	bReady := FALSE;
	nErrorId := BACnet_ERR_OPERATIONAL;
END_IF
(* set error flag *)
bError := (nErrorId <> BACnet_ERR_NO_ERROR);

END_FUNCTION_BLOCK

// POUs/BACnet Objects/Local (Server)/FB_BACnet_Command
FUNCTION_BLOCK FB_BACnet_Command
VAR_INPUT
	bEnablePV		: BOOL;
	nPV				: UDINT;
	bRetrigger		: BOOL; (* execute selected action on raising edge again *)
END_VAR
VAR_IN_OUT
	Device	: FB_BACnet_Device;
END_VAR
VAR_OUTPUT
	bReady			: BOOL;
	nPresentValue	: UDINT;
	bAllWritesOk	: BOOL; (* all actions in selected action list are written *)
	bInProcess		: BOOL; (* object is busy *)
	bError			: BOOL;
	nErrorId		: UINT;
END_VAR
VAR
	_PresentValueIn AT%I*: UDINT; 		(* ~(BACnet_PresentValue 			:		: )
								   			(BACnet_ObjectType 				: CMD	: )	*)
    _PresentValueOut AT%Q*: UDINT;		(* ~(BACnet_PresentValue	 	   	:		: )	*)
	_InProcess AT%I*: BOOL;				(* ~(BACnet_InProcess 				:		: )	*)
	_AllWritesSuccessful AT%I*: BOOL;	(* ~(BACnet_AllWritesSuccessful		:		: )	*)
	_nUpdateCount : UDINT := 0;
	_rtrigRetriggerPv : R_TRIG;
	_bRetriggerReq : BOOL;
END_VAR

(* update server device *)
IF (Device._nUpdateCount = _nUpdateCount) THEN
	Device();
END_IF
(* remind current number of update counter *)
_nUpdateCount := Device._nUpdateCount;

(* call trigger *)
_rtrigRetriggerPv(CLK:= bRetrigger, Q=> );
IF _rtrigRetriggerPv.Q THEN
	_bRetriggerReq := TRUE;
END_IF

IF Device.bFirstCycle THEN
	(* first call of the server device since reboot/reset *)
	bReady := FALSE;
	_PresentValueOut := 0;
	_bRetriggerReq := FALSE;

ELSIF Device.bOperational THEN
	(* ready state *)
	bReady := TRUE;
	nErrorId := BACnet_ERR_NO_ERROR;
	(* activities *)
	bAllWritesOk := _AllWritesSuccessful;
	bInProcess := _InProcess;
	(* present value from BACnet *)
	nPresentValue := _PresentValueIn;
	(* present value to BACnet *)
	IF bEnablePV THEN
		IF (NOT bInProcess) THEN
			IF _bRetriggerReq THEN
				(* trigger action list *)
				_PresentValueOut := 0;
			ELSE
				(* set present value *)
				_PresentValueOut := nPV;
			END_IF
			_bRetriggerReq := FALSE;
		END_IF
	ELSE
		(* deactivate mapped present value --> other clients can write to property *)
		_PresentValueOut := 16#0;
		_bRetriggerReq := FALSE;
	END_IF
ELSE
	(* server device not ready, reset local ready also *)
	bReady := FALSE;
	nErrorId := BACnet_ERR_OPERATIONAL;
	_bRetriggerReq := FALSE;
END_IF
(* set error flag *)
bError := (nErrorId <> BACnet_ERR_NO_ERROR);

END_FUNCTION_BLOCK

// POUs/BACnet Objects/Local (Server)/FB_BACnet_EventEnrollment
FUNCTION_BLOCK FB_BACnet_EventEnrollment
VAR_IN_OUT
	Device					: FB_BACnet_Device;
END_VAR
VAR_OUTPUT
	bReady					: BOOL;
	eEventState				: E_BACNETEVENTSTATE;
	bAckedTrans_ToOffNormal : BOOL;
	bAckedTrans_ToFault		: BOOL;
	bAckedTrans_ToNormal	: BOOL;
	bError					: BOOL;
	nErrorId				: UINT;
END_VAR
VAR
	_EventState AT%I*: WORD; 			(* ~(BACnet_EventState 			:		: )
											(BACnet_ObjectType			: EE	: )	*)
	_AckedTransitions AT%I*: WORD; 		(* ~(BACnet_AckedTransitions 	:		: )	*)
	_AckedTransBits : ST_BACnet_EventTransitionBits;
	_nUpdateCount : UDINT := 0;
END_VAR

(* update server device *)
IF (Device._nUpdateCount = _nUpdateCount) THEN
	Device();
END_IF
(* remind current number of update counter *)
_nUpdateCount := Device._nUpdateCount;

(* check BitString format *)
IF (_AckedTransitions < 5) THEN
	(* wrong mapping *)
	nErrorId := BACnet_ERR_WRONG_MAPPING;
	bReady := FALSE;

ELSIF Device.bOperational THEN
	(* ready state *)
	bReady := TRUE;
	nErrorId := BACnet_ERR_NO_ERROR;

	(* copy states *)
	bAckedTrans_ToOffNormal := _AckedTransBits.to_offnormal;
	bAckedTrans_ToFault := _AckedTransBits.to_fault;
	bAckedTrans_ToNormal := _AckedTransBits.to_normal;
	eEventState := TO_INT(_EventState);

ELSE
	bReady := FALSE;
	nErrorId := BACnet_ERR_OPERATIONAL;
END_IF
(* set error flag *)
bError := (nErrorId <> BACnet_ERR_NO_ERROR);

END_FUNCTION_BLOCK

// POUs/BACnet Objects/Local (Server)/FB_BACnet_File
FUNCTION_BLOCK FB_BACnet_File
VAR_IN_OUT
	Device	: FB_BACnet_Device;
END_VAR
VAR_OUTPUT
	bReady			: BOOL;
	nFileSize		: UDINT;
	bError			: BOOL;
	nErrorId		: UINT;
END_VAR
VAR
	_FileSize 			AT%I*: UDINT; 	(* ~(BACnet_FileSize 				:		: )
					   						(BACnet_ObjectType 				: FILE	: )	*)
	_nUpdateCount		: UDINT := 0;
END_VAR

(* update server device *)
IF (Device._nUpdateCount = _nUpdateCount) THEN
	Device();
END_IF
(* remind current number of update counter *)
_nUpdateCount := Device._nUpdateCount;

IF Device.bOperational THEN
	(* ready state *)
	bReady := TRUE;
	nErrorId := BACnet_ERR_NO_ERROR;
	nFileSize := _FileSize;
ELSE
	(* server device not ready, reset local ready also *)
	bReady := FALSE;
	nErrorId := BACnet_ERR_OPERATIONAL;
END_IF
(* set error flag *)
bError := (nErrorId <> BACnet_ERR_NO_ERROR);

END_FUNCTION_BLOCK

// POUs/BACnet Objects/Local (Server)/FB_BACnet_Group
FUNCTION_BLOCK FB_BACnet_Group
VAR_IN_OUT
	Device	: FB_BACnet_Device;
END_VAR
VAR_OUTPUT
	bReady			: BOOL;
	bError			: BOOL;
	nErrorId		: UINT;
END_VAR
VAR
	_nUpdateCount : UDINT := 0; (* ~(BACNET_OBJECTTYPE : GROUP : NOLINK)	*)
END_VAR

(* update server device *)
IF (Device._nUpdateCount = _nUpdateCount) THEN
	Device();
END_IF
(* remind current number of update counter *)
_nUpdateCount := Device._nUpdateCount;

IF Device.bOperational THEN
	(* ready state *)
	bReady := TRUE;
	nErrorId := BACnet_ERR_NO_ERROR;
ELSE
	(* server device not ready, reset local ready also *)
	bReady := FALSE;
	nErrorId := BACnet_ERR_OPERATIONAL;
END_IF
(* set error flag *)
bError := (nErrorId <> BACnet_ERR_NO_ERROR);

END_FUNCTION_BLOCK

// POUs/BACnet Objects/Local (Server)/FB_BACnet_MultiStateInput
FUNCTION_BLOCK FB_BACnet_MultiStateInput
VAR_IN_OUT
	Device	: FB_BACnet_Device;
END_VAR
VAR_OUTPUT
	bReady			: BOOL;
	nPresentValue	: UDINT;
	bOverridden		: BOOL;
	bOutOfService	: BOOL;
	bFault			: BOOL;
	bInAlarm		: BOOL;
	bError			: BOOL;
	nErrorId		: UINT;
END_VAR
VAR
	_PresentValue AT%I*: UDINT; 	(* ~(BACnet_PresentValue 	:		: )
								   		(BACnet_ObjectType 		: MI	: )	*)
	_StatusFlags AT%I*: WORD; 		(* ~(BACnet_StatusFlags 	:		: )	*)
	_StatusFlagsBits : ST_BACnet_StatusFlags;

	_nUpdateCount : UDINT := 0;
END_VAR

(* update server device *)
IF (Device._nUpdateCount = _nUpdateCount) THEN
	Device();
END_IF
(* remind current number of update counter *)
_nUpdateCount := Device._nUpdateCount;

(* check BitString format of StatusFlags --> if StatusFlags are less than 4, object isn't linked correctly *)
IF (_StatusFlags < 4) THEN
	(* wrong mapping *)
	nErrorId := BACnet_ERR_WRONG_MAPPING;
	bReady := FALSE;

ELSIF Device.bOperational THEN
	(* ready state *)
	bReady := TRUE;
	nErrorId := BACnet_ERR_NO_ERROR;

	(* present value *)
	nPresentValue := _PresentValue;

	(* build bit states *)
	_StatusFlagsBits := F_BACnet_StatusFlags(_StatusFlags);

	(* copy states to output *)
	bOverridden := _StatusFlagsBits.overridden;
	bOutOfService := _StatusFlagsBits.out_of_service;
	bFault := _StatusFlagsBits.fault;
	bInAlarm := _StatusFlagsBits.in_alarm;

ELSE
	(* server device not ready, reset local ready also *)
	bReady := FALSE;
	nErrorId := BACnet_ERR_OPERATIONAL;
END_IF
(* set error flag *)
bError := (nErrorId <> BACnet_ERR_NO_ERROR);

END_FUNCTION_BLOCK

// POUs/BACnet Objects/Local (Server)/FB_BACnet_MultiStateOutput
FUNCTION_BLOCK FB_BACnet_MultiStateOutput
VAR_INPUT
	bEnablePV		: BOOL; (* enable present value with priority x in priority array, FALSE = priority x disable *)
	bNullPV			: BOOL; (* clear priority entry *)
	nPV				: UDINT; (* number for priority x, when input bEnablePV is TRUE *)
END_VAR
VAR_IN_OUT
	Device	: FB_BACnet_Device;
END_VAR
VAR_OUTPUT
	bReady			: BOOL;
	nPresentValue	: UDINT;
	bOverridden		: BOOL;
	bOutOfService	: BOOL;
	bFault			: BOOL;
	bInAlarm		: BOOL;
	nNbrOfStates	: UDINT;
	bError			: BOOL;
	nErrorId		: UINT;
END_VAR
VAR
	_PresentValue AT%I*: UDINT; 			(* ~(BACnet_PresentValue 		:		: )
								   				(BACnet_ObjectType			: MO	: )	*)
	_NumberOfStates AT%I*: UDINT;			(* ~(BACnet_NumberOfStates		:		: )	*)
	_StatusFlags AT%I*: WORD; 				(* ~(BACnet_StatusFlags			:		: )	*)
    _PresentValue_Priority12 AT%Q*: UDINT;	(* ~(BACnet_PresentValue_Priority12:	: )	*)
	_StatusFlagsBits : ST_BACnet_StatusFlags;
	_nUpdateCount : UDINT := 0;
END_VAR

(* update server device *)
IF (Device._nUpdateCount = _nUpdateCount) THEN
	Device();
END_IF
(* remind current number of update counter *)
_nUpdateCount := Device._nUpdateCount;

IF Device.bFirstCycle THEN
	(* first call of the server device since reboot/reset *)
	bReady := FALSE;
	_PresentValue_Priority12 := 16#FFFFFFFF;

ELSIF (_StatusFlags < 4) THEN
	(* wrong mapping *)
	nErrorId := BACnet_ERR_WRONG_MAPPING;
	bReady := FALSE;

ELSIF Device.bOperational THEN
	(* ready state *)
	bReady := TRUE;
	nErrorId := BACnet_ERR_NO_ERROR;

	(* write into priority array *)
	_PresentValue_Priority12 := F_BACnet_MultiStatePV(bEnablePV, bNullPV, nPV);

	(* present value *)
	nPresentValue := _PresentValue;

	(* build bit states *)
	_StatusFlagsBits := F_BACnet_StatusFlags(_StatusFlags);

	(* copy states to output *)
	bOverridden := _StatusFlagsBits.overridden;
	bOutOfService := _StatusFlagsBits.out_of_service;
	bFault := _StatusFlagsBits.fault;
	bInAlarm := _StatusFlagsBits.in_alarm;

	(* number of states *)
	nNbrOfStates := _NumberOfStates;

ELSE
	(* server device not ready, reset local ready also *)
	bReady := FALSE;
	nErrorId := BACnet_ERR_OPERATIONAL;
END_IF
(* set error flag *)
bError := (nErrorId <> BACnet_ERR_NO_ERROR);

END_FUNCTION_BLOCK

// POUs/BACnet Objects/Local (Server)/FB_BACnet_MultiStateValue
FUNCTION_BLOCK FB_BACnet_MultiStateValue
VAR_INPUT
	bEnablePV		: BOOL; (* enable present value with priority x in priority array, FALSE = priority x disable *)
	bNullPV			: BOOL; (* clear priority entry *)
	nPV				: UDINT; (* number for priority x, when input bEnablePV is TRUE *)
END_VAR
VAR_IN_OUT
	Device	: FB_BACnet_Device;
END_VAR
VAR_OUTPUT
	bReady			: BOOL;
	nPresentValue	: UDINT;
	bOverridden		: BOOL;
	bOutOfService	: BOOL;
	bFault			: BOOL;
	bInAlarm		: BOOL;
	nNbrOfStates	: UDINT;
	bError			: BOOL;
	nErrorId		: UINT;
END_VAR
VAR
	_PresentValue AT%I*: UDINT; 			(* ~(BACnet_PresentValue 		:		: )
								   				(BACnet_ObjectType 			: MV	: )	*)
	_NumberOfStates AT%I*: UDINT;			(* ~(BACnet_NumberOfStates		:		: )	*)
	_StatusFlags AT%I*: WORD; 				(* ~(BACnet_StatusFlags 		:		: )	*)
    _PresentValue_Priority12 AT%Q*: UDINT;	(* ~(BACnet_PresentValue_Priority12:	: )	*)
	_nUpdateCount : UDINT := 0;
	_StatusFlagsBits : ST_BACnet_StatusFlags;
END_VAR

(* update server device *)
IF (Device._nUpdateCount = _nUpdateCount) THEN
	Device();
END_IF
(* remind current number of update counter *)
_nUpdateCount := Device._nUpdateCount;

IF Device.bFirstCycle THEN
	(* first call of the server device since reboot/reset *)
	bReady := FALSE;
	_PresentValue_Priority12 := 16#FFFFFFFF;

ELSIF (_StatusFlags < 4) THEN
	(* wrong mapping *)
	nErrorId := BACnet_ERR_WRONG_MAPPING;
	bReady := FALSE;

ELSIF Device.bOperational THEN
	(* ready state *)
	bReady := TRUE;
	nErrorId := BACnet_ERR_NO_ERROR;

	(* write into priority array *)
	_PresentValue_Priority12 := F_BACnet_MultiStatePV(bEnablePV, bNullPV, nPV);

	(* present value *)
	nPresentValue := _PresentValue;

	(* build bit states *)
	_StatusFlagsBits := F_BACnet_StatusFlags(_StatusFlags);

	(* copy states to output *)
	bOverridden := _StatusFlagsBits.overridden;
	bOutOfService := _StatusFlagsBits.out_of_service;
	bFault := _StatusFlagsBits.fault;
	bInAlarm := _StatusFlagsBits.in_alarm;

	(* number of states *)
	nNbrOfStates := _NumberOfStates;

ELSE
	(* server device not ready, reset local ready also *)
	bReady := FALSE;
	nErrorId := BACnet_ERR_OPERATIONAL;
END_IF
(* set error flag *)
bError := (nErrorId <> BACnet_ERR_NO_ERROR);

END_FUNCTION_BLOCK

// POUs/BACnet Objects/Local (Server)/FB_BACnet_NotificationClass
FUNCTION_BLOCK FB_BACnet_NotificationClass
VAR_IN_OUT
	Device	: FB_BACnet_Device;
END_VAR
VAR_OUTPUT
	bReady			: BOOL;
	bError			: BOOL;
	nErrorId		: UINT;
END_VAR
VAR
	_ObjectId AT%I* : DWORD;					(* ~(BACnet_ObjectIdentifier:		: LINK)
													(BACnet_ObjectType		:	NC	: ) *)
	_nUpdateCount	: UDINT := 0;
END_VAR

(* update server device *)
IF (Device._nUpdateCount = _nUpdateCount) THEN
	Device();
END_IF
(* remind current number of update counter *)
_nUpdateCount := Device._nUpdateCount;

IF Device.bOperational THEN
	(* ready state *)
	bReady := TRUE;
	nErrorId := BACnet_ERR_NO_ERROR;
ELSE
	(* server device not ready, reset local ready also *)
	bReady := FALSE;
	nErrorId := BACnet_ERR_OPERATIONAL;
END_IF
(* set error flag *)
bError := (nErrorId <> BACnet_ERR_NO_ERROR);

END_FUNCTION_BLOCK

// POUs/BACnet Objects/Local (Server)/FB_BACnet_PulseConverter
FUNCTION_BLOCK FB_BACnet_PulseConverter
VAR_IN_OUT
	Device			: FB_BACnet_Device;
END_VAR
VAR_OUTPUT
	bReady			: BOOL;
	fPresentValue	: REAL;
	nCount			: UDINT;
	bOverridden		: BOOL;
	bOutOfService	: BOOL;
	bFault			: BOOL;
	bInAlarm		: BOOL;
	bError			: BOOL;
	nErrorId		: UINT;
END_VAR
VAR
	_PresentValueIn AT%I*: REAL; 	(* ~(BACnet_PresentValue 		:		: )
								   		(BACnet_ObjectType 			: PC	: )	*)
	_Count AT%I*: UDINT;			(* ~(BACnet_Count		 		:		: ) *)
	_StatusFlags AT%I*: WORD; 		(* ~(BACnet_StatusFlags 		:		: )	*)
	_StatusFlagsBits : ST_BACnet_StatusFlags;
	_nUpdateCount : UDINT := 0;
END_VAR

(* update server device *)
IF (Device._nUpdateCount = _nUpdateCount) THEN
	Device();
END_IF
(* remind current number of update counter *)
_nUpdateCount := Device._nUpdateCount;

IF Device.bFirstCycle THEN
	(* first call of the server device since reboot/reset *)
	bReady := FALSE;

ELSIF (_StatusFlags < 4) THEN
	(* wrong mapping *)
	nErrorId := BACnet_ERR_WRONG_MAPPING;
	bReady := FALSE;

ELSIF Device.bOperational THEN
	(* ready state *)
	bReady := TRUE;
	nErrorId := BACnet_ERR_NO_ERROR;

	(* present value *)
	fPresentValue := _PresentValueIn;

	(* build bit states *)
	_StatusFlagsBits := F_BACnet_StatusFlags(_StatusFlags);

	(* copy states to output *)
	bOverridden		:= _StatusFlagsBits.overridden;
	bOutOfService	:= _StatusFlagsBits.out_of_service;
	bFault			:= _StatusFlagsBits.fault;
	bInAlarm		:= _StatusFlagsBits.in_alarm;

	(* additional information *)
	nCount			:= _Count;

ELSE
	(* server device not ready, reset local ready flag *)
	bReady := FALSE;
	nErrorId := BACnet_ERR_OPERATIONAL;
END_IF
(* set error flag *)
bError := (nErrorId <> BACnet_ERR_NO_ERROR);

END_FUNCTION_BLOCK

// POUs/BACnet Objects/Local (Server)/FB_BACnet_Schedule
FUNCTION_BLOCK FB_BACnet_Schedule
VAR_IN_OUT
	Device	: FB_BACnet_Device;
END_VAR
VAR_OUTPUT
	bReady			: BOOL;
	bPresentValue	: BOOL;
	bOverridden		: BOOL;
	bOutOfService	: BOOL;
	bFault			: BOOL;
	bInAlarm		: BOOL;
	bError			: BOOL;
	nErrorId		: UINT;
END_VAR
VAR
	_StatusFlags AT%I*: WORD; 	(* ~(BACnet_StatusFlags 				:		: )	*)
	_PresentValue AT%I*: BOOL;	(* ~(BACnet_PresentValueBool 			:		: )
									(BACnet_ObjectType 					: SCHED	: )	*)
	_StatusFlagsBits : ST_BACnet_StatusFlags;
	_nUpdateCount : UDINT := 0;
END_VAR

(* update server device *)
IF (Device._nUpdateCount = _nUpdateCount) THEN
	Device();
END_IF
(* remind current number of update counter *)
_nUpdateCount := Device._nUpdateCount;

(* check BitString format of StatusFlags --> if StatusFlags are less than 4, object isn't linked correctly *)
IF (_StatusFlags < 4) THEN
	(* wrong mapping *)
	nErrorId := BACnet_ERR_WRONG_MAPPING;
	bReady := FALSE;

ELSIF Device.bOperational THEN
	(* ready state *)
	bReady := TRUE;
	nErrorId := BACnet_ERR_NO_ERROR;

	(* present value *)
	bPresentValue := _PresentValue;

	(* build bit states *)
	_StatusFlagsBits := F_BACnet_StatusFlags(_StatusFlags);

	(* copy states to output *)
	bOverridden := _StatusFlagsBits.overridden;
	bOutOfService := _StatusFlagsBits.out_of_service;
	bFault := _StatusFlagsBits.fault;
	bInAlarm := _StatusFlagsBits.in_alarm;

ELSE
	bReady := FALSE;
	nErrorId := BACnet_ERR_OPERATIONAL;
END_IF
(* set error flag *)
bError := (nErrorId <> BACnet_ERR_NO_ERROR);

END_FUNCTION_BLOCK

// POUs/BACnet Objects/Local (Server)/FB_BACnet_TrendLog
FUNCTION_BLOCK FB_BACnet_TrendLog
VAR_IN_OUT
	Device	: FB_BACnet_Device;
END_VAR
VAR_OUTPUT
	bReady			: BOOL;
	bLogEnable		: BOOL;
	nTotalCount		: UDINT;
	bError			: BOOL;
	nErrorId		: UINT;
END_VAR
VAR
	_TotalRecordCount AT%I*: UDINT;	(* ~(BACnet_TotalRecordCount:		: )
										(BACnet_ObjectType		: TLOG	: )	*)
	_LogEnable AT%I*: BOOL;			(* ~(BACnet_LogEnable		: 		: )	*)
	_nUpdateCount : UDINT := 0;
END_VAR

(* update server device *)
IF (Device._nUpdateCount = _nUpdateCount) THEN
	Device();
END_IF
(* remind current number of update counter *)
_nUpdateCount := Device._nUpdateCount;

IF Device.bOperational THEN
	(* ready state *)
	bReady := TRUE;
	nErrorId := BACnet_ERR_NO_ERROR;
	bLogEnable := _LogEnable;

	(* other states *)
	nTotalCount := _TotalRecordCount;

ELSE
	bReady := FALSE;
	nErrorId := BACnet_ERR_OPERATIONAL;
END_IF
(* set error flag *)
bError := (nErrorId <> BACnet_ERR_NO_ERROR);

END_FUNCTION_BLOCK

// POUs/BACnet Objects/Remote (Client)/Extended Process Data/FB_BACnet_RemoteAccumulator_EX
FUNCTION_BLOCK FB_BACnet_RemoteAccumulator_EX
VAR_IN_OUT
	RemoteDevice		: FB_BACnet_RemoteDevice;
END_VAR
VAR_OUTPUT
	bReady				: BOOL;
	nPresentValue		: UDINT;
	bOverridden			: BOOL;
	bOutOfService		: BOOL;
	bFault				: BOOL;
	bInAlarm			: BOOL;
	bOverRange			: BOOL;
	bUnderRange			: BOOL;
	bNoSensor			: BOOL;
	bOpenLoop			: BOOL;
	bCommFailure		: BOOL;
	bShortedLoop		: BOOL;
	bOtherFault			: BOOL;
	tObjectID			: T_BACnet_ObjectIdentifier := 16#FFFFFFFF;
	bError				: BOOL;
	nErrorId			: UINT;
END_VAR
VAR
	_PresentValue AT%I*:UDINT;			(* ~(BACnet_PresentValue				:		: )
											(BACnet_ObjectType					: ACC	: )
											(BACnet_RemoteCycletimeRead			: 1000	: )
											(BACnet_RemoteFlagsRead				: 1		: )
											(BACnet_RemoteResubscriptionInterval: 240	: )
                                			(BACnet_RemoteCycleTimeWrite   		: 1000	: )
                                			(BACnet_RemoteFlagsWrite       		: 1		: )	*)
	_ObjectId AT%I*: DWORD;				(* ~(BACnet_ObjectIdentifier			:		: LINK) *)
	_StatusFlags AT%I*:WORD;			(* ~(BACnet_StatusFlags					:		: )	*)
	_Reliability AT%I*:WORD;			(* ~(BACnet_Reliability					:		: )	*)
	_StatusFlagsBits : ST_BACnet_StatusFlags;

	_nUpdateCount : UDINT := 0;
END_VAR

(* update client device *)
IF RemoteDevice._nUpdateCount = _nUpdateCount THEN
	RemoteDevice();
END_IF
(* remind current number of update counter *)
_nUpdateCount := RemoteDevice._nUpdateCount;

IF NOT RemoteDevice.bOperational THEN
	nErrorId := BACnet_ERR_OPERATIONAL;
	bReady := FALSE;

ELSIF (F_BACnet_GetObjType(_ObjectId) <> BACnetObjectType_Accumulator) THEN
	(* wrong mapping / invalid object ID *)
	IF _ObjectId = 0 THEN
		nErrorId := BACnet_ERR_WRONG_MAPPING;
	ELSE
		nErrorId := BACnet_ERR_INVALID_OBJECTID;
	END_IF
	bReady := FALSE;
	tObjectID := 16#FFFFFFFF;

ELSIF _StatusFlags >= 4 THEN
	(* clear error flag *)
	nErrorId := BACnet_ERR_NO_ERROR;
	bReady := TRUE;
	(* copy present value *)
	nPresentValue := _PresentValue;

	(* build bit states *)
	_StatusFlagsBits := F_BACnet_StatusFlags(_StatusFlags);

	(* copy states to output *)
	bOverridden := _StatusFlagsBits.overridden;
	bOutOfService := _StatusFlagsBits.out_of_service;
	bFault := _StatusFlagsBits.fault;
	bInAlarm := _StatusFlagsBits.in_alarm;
	bOverRange := (_Reliability = TO_WORD(BACnetReliability_over_range));
	bUnderRange := (_Reliability = TO_WORD(BACnetReliability_under_range));
	bNoSensor := (_Reliability = TO_WORD(BACnetReliability_no_sensor));
	bOpenLoop := (_Reliability = TO_WORD(BACnetReliability_open_loop));
	bCommFailure := (_Reliability = TO_WORD(BACnetReliability_communication_failure));
	bShortedLoop := (_Reliability = TO_WORD(BACnetReliability_shorted_loop));
	bOtherFault := (_Reliability = TO_WORD(BACnetReliability_unreliable_other));
	tObjectID := _ObjectId;

ELSE
	bReady := FALSE;
	(* and set error ID *)
	nErrorId := BACnet_ERR_WRONG_MAPPING;
END_IF

(* set error flag *)
bError := (nErrorId <> BACnet_ERR_NO_ERROR);

END_FUNCTION_BLOCK

// POUs/BACnet Objects/Remote (Client)/Extended Process Data/FB_BACnet_RemoteAnalogInput_EX
FUNCTION_BLOCK FB_BACnet_RemoteAnalogInput_EX
VAR_IN_OUT
	RemoteDevice			: FB_BACnet_RemoteDevice;
END_VAR
VAR_OUTPUT
	bReady				: BOOL;
	fPresentValue		: REAL;
	bOverridden			: BOOL;
	bOutOfService		: BOOL;
	bFault				: BOOL;
	bInAlarm			: BOOL;
	bOverRange			: BOOL;
	bUnderRange			: BOOL;
	bNoSensor			: BOOL;
	bOpenLoop			: BOOL;
	bShortedLoop		: BOOL;
	bOtherFault			: BOOL;
	eEventState			: E_BACNETEVENTSTATE;
	tObjectID			: T_BACnet_ObjectIdentifier := 16#FFFFFFFF;
	bError				: BOOL;
	nErrorId			: UINT;
END_VAR
VAR
	_PresentValue AT%I*: REAL; 			(* ~(BACnet_PresentValue 				:		: )
								   			(BACnet_ObjectType 					: AI	: )
											(BACnet_RemoteCycletimeRead 		: 1000	: )
											(BACnet_RemoteFlagsRead        		: 1		: )
											(BACnet_RemoteResubscriptionInterval: 240	: )
	                                		(BACnet_RemoteCycleTimeWrite   		: 1000	: )
	                                		(BACnet_RemoteFlagsWrite       		: 1		: )	*)
	_ObjectId AT%I*: DWORD;				(* ~(BACnet_ObjectIdentifier			:		: LINK) *)
	_StatusFlags AT%I*: WORD; 			(* ~(BACnet_StatusFlags 				:		: )	*)
	_Reliability AT%I*: WORD;; 			(* ~(BACnet_Reliability 				:		: )	*)
	_EventState AT%I*: WORD;			(* ~(BACnet_EventState					:		: )	*)
	_nUpdateCount : UDINT := 0;
	_StatusFlagsBits : ST_BACnet_StatusFlags;
END_VAR

(* update client device *)
IF RemoteDevice._nUpdateCount = _nUpdateCount THEN
	RemoteDevice();
END_IF
(* remind current number of update counter *)
_nUpdateCount := RemoteDevice._nUpdateCount;

IF NOT RemoteDevice.bOperational THEN
	nErrorId := BACnet_ERR_OPERATIONAL;
	bReady := FALSE;

ELSIF (F_BACnet_GetObjType(_ObjectId) <> BACnetObjectType_AnalogInput) THEN
	(* wrong mapping / invalid object ID *)
	IF _ObjectId = 0 THEN
		nErrorId := BACnet_ERR_WRONG_MAPPING;
	ELSE
		nErrorId := BACnet_ERR_INVALID_OBJECTID;
	END_IF
	bReady := FALSE;
	tObjectID := 16#FFFFFFFF;

ELSIF _StatusFlags >= 4 THEN
	(* clear error flag *)
	nErrorId := BACnet_ERR_NO_ERROR;
	(* ready state *)
	bReady := TRUE;

	(* present value *)
	fPresentValue := _PresentValue;

	(* build bit states *)
	_StatusFlagsBits := F_BACnet_StatusFlags(_StatusFlags);

	(* copy states to output *)
	bOverridden := _StatusFlagsBits.overridden;
	bOutOfService := _StatusFlagsBits.out_of_service;
	bFault := _StatusFlagsBits.fault;
	bInAlarm := _StatusFlagsBits.in_alarm;
	bOverRange := (_Reliability = TO_WORD(BACnetReliability_over_range));
	bUnderRange := (_Reliability = TO_WORD(BACnetReliability_under_range));
	bNoSensor := (_Reliability = TO_WORD(BACnetReliability_no_sensor));
	bOpenLoop := (_Reliability = TO_WORD(BACnetReliability_open_loop));
	bShortedLoop := (_Reliability = TO_WORD(BACnetReliability_shorted_loop));
	bOtherFault := (_Reliability = TO_WORD(BACnetReliability_unreliable_other));
	eEventState := TO_INT(_EventState);
	tObjectID := _ObjectId;
ELSE
	(* server device not ready, reset local ready also *)
	bReady := FALSE;
	(* and set error ID *)
	nErrorId := BACnet_ERR_WRONG_MAPPING;
END_IF

(* set error flag *)
bError := (nErrorId <> BACnet_ERR_NO_ERROR);

END_FUNCTION_BLOCK

// POUs/BACnet Objects/Remote (Client)/Extended Process Data/FB_BACnet_RemoteAnalogOutput_EX
FUNCTION_BLOCK FB_BACnet_RemoteAnalogOutput_EX
VAR_INPUT
	bEnablePV			: BOOL; (* enable present value with priority x in priority array, FALSE = priority x disable *)
	bNullPV				: BOOL; (* clear priority entry *)
	fPV					: REAL; (* decimal number for priority x, when input bEnablePV is TRUE *)
END_VAR
VAR_IN_OUT
	RemoteDevice		: FB_BACnet_RemoteDevice;
END_VAR
VAR_OUTPUT
	bReady				: BOOL;
	fPresentValue		: REAL;
	bOverridden			: BOOL;
	bOutOfService		: BOOL;
	bFault				: BOOL;
	bInAlarm			: BOOL;
	bNoOutput			: BOOL;
	bOpenLoop			: BOOL;
	bShortedLoop		: BOOL;
	bOtherFault			: BOOL;
	eEventState			: E_BACNETEVENTSTATE;
	tObjectID			: T_BACnet_ObjectIdentifier := 16#FFFFFFFF;
	bError				: BOOL;
	nErrorId			: UINT;
END_VAR
VAR
	_PresentValue AT%I*: REAL; 			(* ~(BACnet_PresentValue 				:		: )
								   			(BACnet_ObjectType 					: AO	: )
											(BACnet_RemoteCycletimeRead 		: 1000	: )
											(BACnet_RemoteFlagsRead        		: 1		: )
											(BACnet_RemoteResubscriptionInterval: 240	: )
	                                		(BACnet_RemoteCycleTimeWrite   		: 1000	: )
	                                		(BACnet_RemoteFlagsWrite       		: 1		: )	*)
    _PresentValue_Priority12 AT%Q*: DWORD;(* ~(BACnet_PresentValue_Priority12	:		: )	*)
	_ObjectId AT%I*: DWORD;				(* ~(BACnet_ObjectIdentifier			:		: LINK) *)
	_StatusFlags AT%I*: WORD; 			(* ~(BACnet_StatusFlags 				:		: )	*)
	_Reliability AT%I*: WORD;; 			(* ~(BACnet_Reliability 				:		: )	*)
	_EventState AT%I*: WORD;			(* ~(BACnet_EventState					:		: )	*)
	_nUpdateCount : UDINT := 0;
	_StatusFlagsBits : ST_BACnet_StatusFlags;
END_VAR

(* update client device *)
IF RemoteDevice._nUpdateCount = _nUpdateCount THEN
	RemoteDevice();
END_IF
(* remind current number of update counter *)
_nUpdateCount := RemoteDevice._nUpdateCount;

IF RemoteDevice.bFirstCycle THEN
	(* first call of the server device since reboot/reset *)
	bReady := FALSE;
	_PresentValue_Priority12 := F_BACnet_RealNothing();

ELSIF NOT RemoteDevice.bOperational THEN
	nErrorId := BACnet_ERR_OPERATIONAL;
	bReady := FALSE;

ELSIF (F_BACnet_GetObjType(_ObjectId) <> BACnetObjectType_AnalogOutput) THEN
	(* wrong mapping / invalid object ID *)
	IF _ObjectId = 0 THEN
		nErrorId := BACnet_ERR_WRONG_MAPPING;
	ELSE
		nErrorId := BACnet_ERR_INVALID_OBJECTID;
	END_IF
	bReady := FALSE;
	tObjectID := 16#FFFFFFFF;

ELSIF _StatusFlags >= 4 THEN
	(* clear error flag *)
	nErrorId := BACnet_ERR_NO_ERROR;
	(* ready state *)
	bReady := TRUE;

	(* write into priority array *)
	_PresentValue_Priority12 := F_BACnet_RealPV(bEnablePV, bNullPV, fPV);

	(* present value *)
	fPresentValue := _PresentValue;

	(* build bit states *)
	_StatusFlagsBits := F_BACnet_StatusFlags(_StatusFlags);

	(* copy states to output *)
	bOverridden := _StatusFlagsBits.overridden;
	bOutOfService := _StatusFlagsBits.out_of_service;
	bFault := _StatusFlagsBits.fault;
	bInAlarm := _StatusFlagsBits.in_alarm;
	bNoOutput := (_Reliability = TO_WORD(BACnetReliability_no_output));
	bOpenLoop := (_Reliability = TO_WORD(BACnetReliability_open_loop));
	bShortedLoop := (_Reliability = TO_WORD(BACnetReliability_shorted_loop));
	bOtherFault := (_Reliability = TO_WORD(BACnetReliability_unreliable_other));
	eEventState := TO_INT(_EventState);
	tObjectID := _ObjectId;
ELSE
	(* server device not ready, reset local ready also *)
	bReady := FALSE;
	(* and set error ID *)
	nErrorId := BACnet_ERR_WRONG_MAPPING;
END_IF

(* set error flag *)
bError := (nErrorId <> BACnet_ERR_NO_ERROR);

END_FUNCTION_BLOCK

// POUs/BACnet Objects/Remote (Client)/Extended Process Data/FB_BACnet_RemoteAnalogValue_EX
FUNCTION_BLOCK FB_BACnet_RemoteAnalogValue_EX
VAR_INPUT
	bEnablePV			: BOOL; (* enable present value with priority x in priority array, FALSE = priority x disable *)
	bNullPV				: BOOL; (* clear priority entry *)
	fPV					: REAL; (* decimal number for priority x, when input bEnablePV is TRUE *)
END_VAR
VAR_IN_OUT
	RemoteDevice		: FB_BACnet_RemoteDevice;
END_VAR
VAR_OUTPUT
	bReady				: BOOL;
	fPresentValue		: REAL;
	bOverridden			: BOOL;
	bOutOfService		: BOOL;
	bFault				: BOOL;
	bInAlarm			: BOOL;
	bOverRange			: BOOL;
	bUnderRange			: BOOL;
	bOtherFault			: BOOL;
	eEventState			: E_BACNETEVENTSTATE;
	tObjectID			: T_BACnet_ObjectIdentifier := 16#FFFFFFFF;
	bError				: BOOL;
	nErrorId			: UINT;
END_VAR
VAR
	_PresentValue AT%I*: REAL; 			(* ~(BACnet_PresentValue 				:		: )
								   			(BACnet_ObjectType 					: AV	: )
											(BACnet_RemoteCycletimeRead 		: 1000	: )
											(BACnet_RemoteFlagsRead        		: 1		: )
											(BACnet_RemoteResubscriptionInterval: 240	: )
	                                		(BACnet_RemoteCycleTimeWrite   		: 1000	: )
	                                		(BACnet_RemoteFlagsWrite       		: 1		: )	*)
    _PresentValue_Priority12 AT%Q*: DWORD;(* ~(BACnet_PresentValue_Priority12	:		: )	*)
	_ObjectId AT%I*: DWORD;				(* ~(BACnet_ObjectIdentifier			:		: LINK) *)
	_StatusFlags AT%I*: WORD; 			(* ~(BACnet_StatusFlags 				:		: )	*)
	_Reliability AT%I*: WORD;;			(* ~(BACnet_Reliability 				:		: )	*)
	_EventState AT%I*: WORD;			(* ~(BACnet_EventState					:		: )	*)
	_nUpdateCount : UDINT := 0;
	_StatusFlagsBits : ST_BACnet_StatusFlags;
END_VAR

(* update client device *)
IF RemoteDevice._nUpdateCount = _nUpdateCount THEN
	RemoteDevice();
END_IF
(* remind current number of update counter *)
_nUpdateCount := RemoteDevice._nUpdateCount;

IF RemoteDevice.bFirstCycle THEN
	(* first call of the server device since reboot/reset *)
	bReady := FALSE;
	_PresentValue_Priority12 := F_BACnet_RealNothing();
ELSIF NOT RemoteDevice.bOperational THEN
	nErrorId := BACnet_ERR_OPERATIONAL;
	bReady := FALSE;

ELSIF (F_BACnet_GetObjType(_ObjectId) <> BACnetObjectType_AnalogValue) THEN
	(* wrong mapping / invalid object ID *)
	IF _ObjectId = 0 THEN
		nErrorId := BACnet_ERR_WRONG_MAPPING;
	ELSE
		nErrorId := BACnet_ERR_INVALID_OBJECTID;
	END_IF
	bReady := FALSE;
	tObjectID := 16#FFFFFFFF;

ELSIF _StatusFlags >= 4 THEN
	(* clear error flag *)
	nErrorId := BACnet_ERR_NO_ERROR;
	(* ready state *)
	bReady := TRUE;

	(* write into priority array *)
	_PresentValue_Priority12 := F_BACnet_RealPV(bEnablePV, bNullPV, fPV);

	(* present value *)
	fPresentValue := _PresentValue;

	(* build bit states *)
	_StatusFlagsBits := F_BACnet_StatusFlags(_StatusFlags);

	(* copy states to output *)
	bOverridden := _StatusFlagsBits.overridden;
	bOutOfService := _StatusFlagsBits.out_of_service;
	bFault := _StatusFlagsBits.fault;
	bInAlarm := _StatusFlagsBits.in_alarm;
	bOverRange := (_Reliability = TO_WORD(BACnetReliability_over_range));
	bUnderRange := (_Reliability = TO_WORD(BACnetReliability_under_range));
	bOtherFault := (_Reliability = TO_WORD(BACnetReliability_unreliable_other));
	eEventState := TO_INT(_EventState);
	tObjectID := _ObjectId;
ELSE
	(* server device not ready, reset local ready also *)
	bReady := FALSE;
	(* and set error ID *)
	nErrorId := BACnet_ERR_WRONG_MAPPING;
END_IF

(* set error flag *)
bError := (nErrorId <> BACnet_ERR_NO_ERROR);

END_FUNCTION_BLOCK

// POUs/BACnet Objects/Remote (Client)/Extended Process Data/FB_BACnet_RemoteAveraging_EX
FUNCTION_BLOCK FB_BACnet_RemoteAveraging_EX
VAR_IN_OUT
	RemoteDevice		: FB_BACnet_RemoteDevice;
END_VAR
VAR_OUTPUT
	bReady				: BOOL;
	nAverageValue		: REAL;
	tObjectID			: T_BACnet_ObjectIdentifier := 16#FFFFFFFF;
	bError				: BOOL;
	nErrorId			: UINT;
END_VAR
VAR
	_AverageValue AT%I*: REAL; 		(* ~(BACnet_AverageValue 				:		: )
										(BACnet_ObjectType					: AVG  	: )
										(BACnet_RemoteCycletimeRead 		: 1000	: )
										(BACnet_RemoteFlagsRead        		: 1		: )
										(BACnet_RemoteResubscriptionInterval: 240	: )
										(BACnet_RemoteCycleTimeWrite   		: 1000	: )
										(BACnet_RemoteFlagsWrite       		: 1		: )	*)
	_ObjectId AT%I*: DWORD;			(* ~(BACnet_ObjectIdentifier			:		: LINK) *)

	_nUpdateCount : UDINT := 0;
END_VAR

(* update client device *)
IF RemoteDevice._nUpdateCount = _nUpdateCount THEN
	RemoteDevice();
END_IF
(* remind current number of update counter *)
_nUpdateCount := RemoteDevice._nUpdateCount;

IF NOT RemoteDevice.bOperational THEN
	(* server device not ready, reset local ready also *)
	bReady := FALSE;
	(* and set error ID *)
	nErrorId := BACnet_ERR_OPERATIONAL;

ELSIF (F_BACnet_GetObjType(_ObjectId) <> BACnetObjectType_Averaging) THEN
	(* wrong mapping / invalid object ID *)
	IF _ObjectId = 0 THEN
		nErrorId := BACnet_ERR_WRONG_MAPPING;
	ELSE
		nErrorId := BACnet_ERR_INVALID_OBJECTID;
	END_IF
	bReady := FALSE;
	tObjectID := 16#FFFFFFFF;

ELSE
	(* clear error flag *)
	nErrorId := BACnet_ERR_NO_ERROR;
	(* ready state *)
	bReady := TRUE;
	(* present value *)
	nAverageValue := _AverageValue;
	tObjectID := _ObjectId;

END_IF

(* set error flag *)
bError := (nErrorId <> BACnet_ERR_NO_ERROR);

END_FUNCTION_BLOCK

// POUs/BACnet Objects/Remote (Client)/Extended Process Data/FB_BACnet_RemoteBinaryInput_EX
FUNCTION_BLOCK FB_BACnet_RemoteBinaryInput_EX
VAR_OUTPUT
	bReady				: BOOL;
	bPresentValue		: BOOL;
	bOverridden			: BOOL;
	bOutOfService		: BOOL;
	bFault				: BOOL;
	bInAlarm			: BOOL;
	bNoSensor			: BOOL;
	bOpenLoop			: BOOL;
	bShortedLoop		: BOOL;
	bOtherFault			: BOOL;
	eEventState			: E_BACNETEVENTSTATE;
	nChangeOfState		: UDINT;
	tObjectID			: T_BACnet_ObjectIdentifier := 16#FFFFFFFF;
	bError				: BOOL;
	nErrorId			: UINT;
END_VAR
VAR_IN_OUT
	RemoteDevice			: FB_BACnet_RemoteDevice;
END_VAR
VAR
	_ChangeOfStateCount AT%I*: UDINT;	(* ~(BACnet_ChangeOfStateCount			:		: ) *)
	_ObjectId AT%I*: DWORD;				(* ~(BACnet_ObjectIdentifier			:		: LINK) *)
	_PresentValue AT%I*: WORD; 			(* ~(BACnet_PresentValue 				:		: )
											(BACnet_ObjectType					: BI    : )
											(BACnet_RemoteCycletimeRead 		: 1000	: )
											(BACnet_RemoteFlagsRead        		: 1		: )
											(BACnet_RemoteResubscriptionInterval: 240	: )
		                                	(BACnet_RemoteCycleTimeWrite   		: 1000	: )
		                                	(BACnet_RemoteFlagsWrite       		: 1		: )	*)
	_StatusFlags AT%I*: WORD; 			(* ~(BACnet_StatusFlags 				:	    : )	*)
	_Reliability AT%I*: WORD;; 			(* ~(BACnet_Reliability 				:		: )	*)
	_EventState AT%I*: WORD;			(* ~(BACnet_EventState					:		: )	*)
	_nUpdateCount : UDINT := 0;
	_StatusFlagsBits : ST_BACnet_StatusFlags;
END_VAR

(* update client device *)
IF RemoteDevice._nUpdateCount = _nUpdateCount THEN
	RemoteDevice();
END_IF
(* remind current number of update counter *)
_nUpdateCount := RemoteDevice._nUpdateCount;

IF NOT RemoteDevice.bOperational THEN
	nErrorId := BACnet_ERR_OPERATIONAL;
	bReady := FALSE;

ELSIF (F_BACnet_GetObjType(_ObjectId) <> BACnetObjectType_BinaryInput) THEN
	(* wrong mapping / invalid object ID *)
	IF _ObjectId = 0 THEN
		nErrorId := BACnet_ERR_WRONG_MAPPING;
	ELSE
		nErrorId := BACnet_ERR_INVALID_OBJECTID;
	END_IF
	bReady := FALSE;
	tObjectID := 16#FFFFFFFF;

ELSIF _StatusFlags >= 4 THEN
	(* clear error flag *)
	nErrorId := BACnet_ERR_NO_ERROR;
	(* ready state *)
	bReady := TRUE;

	(* present value *)
	bPresentValue := F_BinPV_To_Bool(TO_INT(_PresentValue));

	(* build bit states *)
	_StatusFlagsBits := F_BACnet_StatusFlags(_StatusFlags);

	(* copy states to output *)
	bOverridden := _StatusFlagsBits.overridden;
	bOutOfService := _StatusFlagsBits.out_of_service;
	bFault := _StatusFlagsBits.fault;
	bInAlarm := _StatusFlagsBits.in_alarm;
	bNoSensor := (_Reliability = TO_WORD(BACnetReliability_no_sensor));
	bOpenLoop := (_Reliability = TO_WORD(BACnetReliability_open_loop));
	bShortedLoop := (_Reliability = TO_WORD(BACnetReliability_shorted_loop));
	bOtherFault := (_Reliability = TO_WORD(BACnetReliability_unreliable_other));
	eEventState := TO_INT(_EventState);
	tObjectID := _ObjectId;

	(* copy change_of_state_count *)
	nChangeOfState := _ChangeOfStateCount;

ELSE
	bReady := FALSE;
	(* and set error ID *)
	nErrorId := BACnet_ERR_WRONG_MAPPING;
END_IF

(* set error flag *)
bError := (nErrorId <> BACnet_ERR_NO_ERROR);

END_FUNCTION_BLOCK

// POUs/BACnet Objects/Remote (Client)/Extended Process Data/FB_BACnet_RemoteBinaryOutput_EX
FUNCTION_BLOCK FB_BACnet_RemoteBinaryOutput_EX
VAR_INPUT
	bEnablePV			: BOOL; (* enable present value with priority x in priority array, FALSE = priority x disable *)
	bNullPV				: BOOL; (* clear priority entry *)
	bPV					: BOOL; (* present value bool type *)
END_VAR
VAR_IN_OUT
	RemoteDevice		: FB_BACnet_RemoteDevice;
END_VAR
VAR_OUTPUT
	bReady				: BOOL;
	bPresentValue		: BOOL;
	bOverridden			: BOOL;
	bOutOfService		: BOOL;
	bFault				: BOOL;
	bInAlarm			: BOOL;
	bNoOutput			: BOOL;
	bOpenLoop			: BOOL;
	bShortedLoop		: BOOL;
	bOtherFault			: BOOL;
	eEventState			: E_BACNETEVENTSTATE;
	nChangeOfState		: UDINT;
	tObjectID			: T_BACnet_ObjectIdentifier := 16#FFFFFFFF;
	bError				: BOOL;
	nErrorId			: UINT;
END_VAR
VAR
	_ChangeOfStateCount AT%I*: UDINT;	(* ~(BACnet_ChangeOfStateCount			:		: ) *)
	_ObjectId AT%I*: DWORD;				(* ~(BACnet_ObjectIdentifier			:		: LINK) *)
	_PresentValue AT%I*: WORD; 			(* ~(BACnet_PresentValue 				:		: )
								   			(BACnet_ObjectType 					: BO	: )
											(BACnet_RemoteCycletimeRead 		: 1000	: )
											(BACnet_RemoteFlagsRead        		: 1		: )
											(BACnet_RemoteResubscriptionInterval: 240	: )
		                            		(BACnet_RemoteCycleTimeWrite   		: 1000	: )
		                            		(BACnet_RemoteFlagsWrite       		: 1		: )	*)
	_StatusFlags AT%I*: WORD; 			(* ~(BACnet_StatusFlags 				:		: )	*)
	_Reliability AT%I*: WORD;;			(* ~(BACnet_Reliability 				:		: )	*)
	_EventState AT%I*: WORD;			(* ~(BACnet_EventState					:		: )	*)
    _PresentValue_Priority12 AT%Q*: WORD;(* ~(BACnet_PresentValue_Priority12	:		: )	*)
	_nUpdateCount : UDINT := 0;
	_StatusFlagsBits : ST_BACnet_StatusFlags;
END_VAR

(* update client device *)
IF RemoteDevice._nUpdateCount = _nUpdateCount THEN
	RemoteDevice();
END_IF
(* remind current number of update counter *)
_nUpdateCount := RemoteDevice._nUpdateCount;

IF RemoteDevice.bFirstCycle THEN
	(* first call of the server device since reboot/reset *)
	bReady := FALSE;
	_PresentValue_Priority12 := TO_WORD(BACnetBinaryPV_Nothing);
ELSIF NOT RemoteDevice.bOperational THEN
	nErrorId := BACnet_ERR_OPERATIONAL;
	bReady := FALSE;

ELSIF (F_BACnet_GetObjType(_ObjectId) <> BACnetObjectType_BinaryOutput) THEN
	(* wrong mapping / invalid object ID *)
	IF _ObjectId = 0 THEN
		nErrorId := BACnet_ERR_WRONG_MAPPING;
	ELSE
		nErrorId := BACnet_ERR_INVALID_OBJECTID;
	END_IF
	bReady := FALSE;
	tObjectID := 16#FFFFFFFF;

ELSIF _StatusFlags >= 4 THEN
	(* clear error flag *)
	nErrorId := BACnet_ERR_NO_ERROR;
	(* ready state *)
	bReady := TRUE;

	(* write into priority array *)
	_PresentValue_Priority12 := TO_WORD(F_Bool_To_BinPV(bEnablePV, bNullPV, bPV));

	(* present value *)
	bPresentValue := F_BinPV_To_Bool(TO_INT(_PresentValue));

	(* build bit states *)
	_StatusFlagsBits := F_BACnet_StatusFlags(_StatusFlags);

	(* copy states to output *)
	bOverridden := _StatusFlagsBits.overridden;
	bOutOfService := _StatusFlagsBits.out_of_service;
	bFault := _StatusFlagsBits.fault;
	bInAlarm := _StatusFlagsBits.in_alarm;
	bNoOutput := (_Reliability = TO_WORD(BACnetReliability_no_output));
	bOpenLoop := (_Reliability = TO_WORD(BACnetReliability_open_loop));
	bShortedLoop := (_Reliability = TO_WORD(BACnetReliability_shorted_loop));
	bOtherFault := (_Reliability = TO_WORD(BACnetReliability_unreliable_other));
	eEventState := TO_INT(_EventState);
	tObjectID := _ObjectId;

	(* copy change_of_state_count *)
	nChangeOfState := _ChangeOfStateCount;
ELSE
	(* server device not ready, reset local ready also *)
	bReady := FALSE;
	(* and set error ID *)
	nErrorId := BACnet_ERR_WRONG_MAPPING;
END_IF

(* set error flag *)
bError := (nErrorId <> BACnet_ERR_NO_ERROR);

END_FUNCTION_BLOCK

// POUs/BACnet Objects/Remote (Client)/Extended Process Data/FB_BACnet_RemoteBinaryValue_EX
FUNCTION_BLOCK FB_BACnet_RemoteBinaryValue_EX
VAR_INPUT
	bEnablePV			: BOOL; (* enable present value with priority x in priority array, FALSE = priority x disable *)
	bNullPV				: BOOL; (* clear priority entry *)
	bPV					: BOOL; (* present value bool type *)
END_VAR
VAR_IN_OUT
	RemoteDevice		: FB_BACnet_RemoteDevice;
END_VAR
VAR_OUTPUT
	bReady				: BOOL;
	bPresentValue		: BOOL;
	bOverridden			: BOOL;
	bOutOfService		: BOOL;
	bFault				: BOOL;
	bInAlarm			: BOOL;
	bOtherFault			: BOOL;
	eEventState			: E_BACNETEVENTSTATE;
	nChangeOfState		: UDINT;
	tObjectID			: T_BACnet_ObjectIdentifier := 16#FFFFFFFF;
	bError				: BOOL;
	nErrorId			: UINT;
END_VAR
VAR
	_ChangeOfStateCount AT%I*: UDINT;	(* ~(BACnet_ChangeOfStateCount			:		: ) *)
	_ObjectId AT%I*: DWORD;				(* ~(BACnet_ObjectIdentifier			:		: LINK) *)
	_PresentValue AT%I*: WORD; 			(* ~(BACnet_PresentValue 				:		: )
								   			(BACnet_ObjectType 					: BV	: )
											(BACnet_RemoteCycletimeRead 		: 1000	: )
											(BACnet_RemoteFlagsRead        		: 1		: )
											(BACnet_RemoteResubscriptionInterval: 240	: )
	                                		(BACnet_RemoteCycleTimeWrite   		: 1000	: )
	                                		(BACnet_RemoteFlagsWrite       		: 1		: )	*)
	_StatusFlags AT%I*: WORD; 			(* ~(BACnet_StatusFlags 				:		: )	*)
	_Reliability AT%I*: WORD;;			(* ~(BACnet_Reliability 				:		: )	*)
	_EventState AT%I*: WORD;			(* ~(BACnet_EventState					:		: )	*)
    _PresentValue_Priority12 AT%Q*: WORD;(* ~(BACnet_PresentValue_Priority12	:		: )	*)
	_nUpdateCount : UDINT := 0;
	_StatusFlagsBits : ST_BACnet_StatusFlags;
END_VAR

(* update client device *)
IF RemoteDevice._nUpdateCount = _nUpdateCount THEN
	RemoteDevice();
END_IF
(* remind current number of update counter *)
_nUpdateCount := RemoteDevice._nUpdateCount;

IF RemoteDevice.bFirstCycle THEN
	(* first call of the server device since reboot/reset *)
	bReady := FALSE;
	_PresentValue_Priority12 := to_word(BACnetBinaryPV_Nothing);
ELSIF NOT RemoteDevice.bOperational THEN
	nErrorId := BACnet_ERR_OPERATIONAL;
	bReady := FALSE;

ELSIF (F_BACnet_GetObjType(_ObjectId) <> BACnetObjectType_BinaryValue) THEN
	(* wrong mapping / invalid object ID *)
	IF _ObjectId = 0 THEN
		nErrorId := BACnet_ERR_WRONG_MAPPING;
	ELSE
		nErrorId := BACnet_ERR_INVALID_OBJECTID;
	END_IF
	bReady := FALSE;
	tObjectID := 16#FFFFFFFF;

ELSIF _StatusFlags >= 4 THEN
	(* clear error flag *)
	nErrorId := BACnet_ERR_NO_ERROR;
	(* ready state *)
	bReady := TRUE;

	(* write into priority array *)
	_PresentValue_Priority12 := TO_WORD(F_Bool_To_BinPV(bEnablePV, bNullPV, bPV));

	(* present value *)
	bPresentValue := F_BinPV_To_Bool(TO_INT(_PresentValue));

	(* build bit states *)
	_StatusFlagsBits := F_BACnet_StatusFlags(_StatusFlags);

	(* copy states to output *)
	bOverridden := _StatusFlagsBits.overridden;
	bOutOfService := _StatusFlagsBits.out_of_service;
	bFault := _StatusFlagsBits.fault;
	bInAlarm := _StatusFlagsBits.in_alarm;
	bOtherFault := (_Reliability = TO_WORD(BACnetReliability_unreliable_other));
	eEventState := TO_INT(_EventState);
	tObjectID := _ObjectId;

	(* copy change_of_state_count *)
	nChangeOfState := _ChangeOfStateCount;

ELSE
	(* server device not ready, reset local ready also *)
	bReady := FALSE;
	(* and set error ID *)
	nErrorId := BACnet_ERR_WRONG_MAPPING;
END_IF

(* set error flag *)
bError := (nErrorId <> BACnet_ERR_NO_ERROR);

END_FUNCTION_BLOCK

// POUs/BACnet Objects/Remote (Client)/Extended Process Data/FB_BACnet_RemoteCalendar_EX
FUNCTION_BLOCK FB_BACnet_RemoteCalendar_EX
VAR_IN_OUT
	RemoteDevice		: FB_BACnet_RemoteDevice;
END_VAR
VAR_OUTPUT
	bReady				: BOOL;
	bPresentValue		: BOOL;
	tObjectID			: T_BACnet_ObjectIdentifier := 16#FFFFFFFF;
	bError				: BOOL;
	nErrorId			: UINT;
END_VAR
VAR
	_PresentValue AT%I*: BOOL;	(* ~(BACnet_PresentValue 				:		: )
									(BACnet_ObjectType 					: CAL	: )
									(BACnet_RemoteCycletimeRead 		: 1000	: )
									(BACnet_RemoteFlagsRead        		: 1		: )
									(BACnet_RemoteResubscriptionInterval: 240	: )
                            		(BACnet_RemoteCycleTimeWrite   		: 1000	: )
                            		(BACnet_RemoteFlagsWrite       		: 1		: )	*)
	_ObjectId AT%I*: DWORD;		(* ~(BACnet_ObjectIdentifier			:		: LINK) *)
	_nUpdateCount : UDINT := 0;
END_VAR

(* update client device *)
IF RemoteDevice._nUpdateCount = _nUpdateCount THEN
	RemoteDevice();
END_IF
(* remind current number of update counter *)
_nUpdateCount := RemoteDevice._nUpdateCount;

IF NOT RemoteDevice.bOperational THEN
	nErrorId := BACnet_ERR_OPERATIONAL;
	bReady := FALSE;

ELSIF (F_BACnet_GetObjType(_ObjectId) <> BACnetObjectType_Calendar) THEN
	(* wrong mapping / invalid object ID *)
	IF _ObjectId = 0 THEN
		nErrorId := BACnet_ERR_WRONG_MAPPING;
	ELSE
		nErrorId := BACnet_ERR_INVALID_OBJECTID;
	END_IF
	bReady := FALSE;
	tObjectID := 16#FFFFFFFF;

ELSE
	(* clear error flag *)
	nErrorId := BACnet_ERR_NO_ERROR;
	(* ready state *)
	bReady := TRUE;
	(* present value *)
	bPresentValue := _PresentValue;
	tObjectID := _ObjectId;

END_IF

(* set error flag *)
bError := (nErrorId <> BACnet_ERR_NO_ERROR);

END_FUNCTION_BLOCK

// POUs/BACnet Objects/Remote (Client)/Extended Process Data/FB_BACnet_RemoteCommand_EX
FUNCTION_BLOCK FB_BACnet_RemoteCommand_EX
VAR_INPUT
	bEnablePV			: BOOL;
	nPV					: UDINT;
	bRetrigger			: BOOL; (* execute selected action on raising edge again *)
END_VAR
VAR_IN_OUT
	RemoteDevice		: FB_BACnet_RemoteDevice;
END_VAR
VAR_OUTPUT
	bReady				: BOOL;
	nPresentValue		: UDINT;
	bAllWritesOk		: BOOL; (* all actions in selected action list are written *)
	bInProcess			: BOOL; (* object is busy *)
	tObjectID			: T_BACnet_ObjectIdentifier := 16#FFFFFFFF;
	bError				: BOOL;
	nErrorId			: UINT;
END_VAR
VAR
	_PresentValueIn AT%I*: UDINT; 		(* ~(BACnet_PresentValue 				:		: )
								   			(BACnet_ObjectType 					: CMD	: )
											(BACnet_RemoteCycletimeRead 		: 1000	: )
											(BACnet_RemoteFlagsRead        		: 1		: )
											(BACnet_RemoteResubscriptionInterval: 240	: )
	                                		(BACnet_RemoteCycleTimeWrite   		: 1000	: )
	                                		(BACnet_RemoteFlagsWrite       		: 1		: )	*)
	_ObjectId AT%I*: DWORD;				(* ~(BACnet_ObjectIdentifier			:		: LINK) *)
	_InProcess AT%I*: BOOL;				(* ~(BACnet_InProcess 					:		: )	*)
	_AllWritesSuccessful AT%I*: BOOL;	(* ~(BACnet_AllWritesSuccessful			:		: )	*)
    _PresentValueOut AT%Q*: UDINT;		(* ~(BACnet_PresentValue	 	   		:      	: )	*)
	_nUpdateCount : UDINT := 0;
	_rtrigRetriggerPv : R_TRIG;
	_bRetriggerReq : BOOL;
END_VAR

(* update client device *)
IF RemoteDevice._nUpdateCount = _nUpdateCount THEN
	RemoteDevice();
END_IF
(* remind current number of update counter *)
_nUpdateCount := RemoteDevice._nUpdateCount;

(* call trigger *)
_rtrigRetriggerPv(CLK:= bRetrigger, Q=> );

IF RemoteDevice.bFirstCycle THEN
	(* first call of the server device since reboot/reset *)
	bReady := FALSE;
	_PresentValueOut := 0;
	_bRetriggerReq := FALSE;

ELSIF NOT RemoteDevice.bOperational THEN
	(* server device not ready, reset local ready also *)
	bReady := FALSE;
	(* and set error ID *)
	nErrorId := BACnet_ERR_WRONG_MAPPING;
	_bRetriggerReq := FALSE;

ELSIF (F_BACnet_GetObjType(_ObjectId) <> BACnetObjectType_Command) THEN
	(* wrong mapping / invalid object ID *)
	IF _ObjectId = 0 THEN
		nErrorId := BACnet_ERR_WRONG_MAPPING;
	ELSE
		nErrorId := BACnet_ERR_INVALID_OBJECTID;
	END_IF
	bReady := FALSE;
	tObjectID := 16#FFFFFFFF;
	_bRetriggerReq := FALSE;

ELSE
	(* object ID *)
	tObjectID := _ObjectId;
	(* clear error flag *)
	nErrorId := BACnet_ERR_NO_ERROR;
	(* activities *)
	bAllWritesOk := _AllWritesSuccessful;
	bInProcess := _InProcess;
	(* ready state *)
	bReady := TRUE;
	(* present value from BACnet *)
	nPresentValue := _PresentValueIn;
	(* present value to BACnet *)
	IF bEnablePV THEN
		IF (NOT bInProcess) THEN
			IF _bRetriggerReq THEN
				(* trigger action list *)
				_PresentValueOut := 0;
			ELSE
				(* set present value *)
				_PresentValueOut := nPV;
			END_IF
			_bRetriggerReq := FALSE;
		END_IF
	ELSE
		(* deactivate mapped present value --> other objects can write to property *)
		_PresentValueOut := 16#0;
		_bRetriggerReq := FALSE;
	END_IF

END_IF

(* set error flag *)
bError := (nErrorId <> BACnet_ERR_NO_ERROR);

END_FUNCTION_BLOCK

// POUs/BACnet Objects/Remote (Client)/Extended Process Data/FB_BACnet_RemoteEventEnrollment_EX
FUNCTION_BLOCK FB_BACnet_RemoteEventEnrollment_EX
VAR_IN_OUT
	RemoteDevice		: FB_BACnet_RemoteDevice;
END_VAR
VAR_OUTPUT
	bReady				: BOOL;
	tObjectID			: T_BACnet_ObjectIdentifier := 16#FFFFFFFF;
	bError				: BOOL;
	nErrorId			: UINT;
END_VAR
VAR
	_ObjectId AT%I*: DWORD;	(* ~(BACnet_ObjectIdentifier:		: LINK)
								(BACNET_OBJECTTYPE		: EE	: ) *)
	_nUpdateCount : UDINT := 0;
END_VAR

(* update client device *)
IF RemoteDevice._nUpdateCount = _nUpdateCount THEN
	RemoteDevice();
END_IF
(* remind current number of update counter *)
_nUpdateCount := RemoteDevice._nUpdateCount;

IF NOT RemoteDevice.bOperational THEN
	(* server device not ready, reset local ready also *)
	bReady := FALSE;
	(* and set error ID *)
	nErrorId := BACnet_ERR_OPERATIONAL;

ELSIF (F_BACnet_GetObjType(_ObjectId) <> BACnetObjectType_EventEnrollment) THEN
	(* wrong mapping / invalid object ID *)
	IF _ObjectId = 0 THEN
		nErrorId := BACnet_ERR_WRONG_MAPPING;
	ELSE
		nErrorId := BACnet_ERR_INVALID_OBJECTID;
	END_IF
	bReady := FALSE;
	tObjectID := 16#FFFFFFFF;

ELSE
	(* clear error flag *)
	nErrorId := BACnet_ERR_NO_ERROR;
	(* ready state *)
	bReady := TRUE;
	tObjectID := _ObjectId;

END_IF

(* set error flag *)
bError := (nErrorId <> BACnet_ERR_NO_ERROR);

END_FUNCTION_BLOCK

// POUs/BACnet Objects/Remote (Client)/Extended Process Data/FB_BACnet_RemoteFile_EX
FUNCTION_BLOCK FB_BACnet_RemoteFile_EX
VAR_IN_OUT
	RemoteDevice		: FB_BACnet_RemoteDevice;
END_VAR
VAR_OUTPUT
	bReady				: BOOL;
	fFileSize			: UDINT;
	tObjectID			: T_BACnet_ObjectIdentifier := 16#FFFFFFFF;
	bError				: BOOL;
	nErrorId			: UINT;
END_VAR
VAR
	_FileSize 			AT%I*: UDINT; 	(* ~(BACnet_FileSize 					:		: )
					   						(BACnet_ObjectType 					: FILE	: )
											(BACnet_RemoteCycletimeRead 		: 1000	: )
											(BACnet_RemoteFlagsRead        		: 1		: )
											(BACnet_RemoteResubscriptionInterval: 240	: )
	                                		(BACnet_RemoteCycleTimeWrite   		: 1000	: )
	                                		(BACnet_RemoteFlagsWrite       		: 1		: )	*)
	_ObjectId AT%I*: DWORD;				(* ~(BACnet_ObjectIdentifier			:		: LINK) *)
	_nUpdateCount		: UDINT := 0;
END_VAR

(* update client device *)
IF RemoteDevice._nUpdateCount = _nUpdateCount THEN
	RemoteDevice();
END_IF
(* remind current number of update counter *)
_nUpdateCount := RemoteDevice._nUpdateCount;

IF NOT RemoteDevice.bOperational THEN
	(* server device not ready, reset local ready also *)
	bReady := FALSE;
	(* and set error ID *)
	nErrorId := BACnet_ERR_OPERATIONAL;

ELSIF (F_BACnet_GetObjType(_ObjectId) <> BACnetObjectType_File) THEN
	(* wrong mapping / invalid object ID *)
	IF _ObjectId = 0 THEN
		nErrorId := BACnet_ERR_WRONG_MAPPING;
	ELSE
		nErrorId := BACnet_ERR_INVALID_OBJECTID;
	END_IF
	bReady := FALSE;
	tObjectID := 16#FFFFFFFF;

ELSE
	(* clear error flag *)
	nErrorId := BACnet_ERR_NO_ERROR;
	(* ready state *)
	bReady := TRUE;
	fFileSize := _FileSize;
	tObjectID := _ObjectId;

END_IF

(* set error flag *)
bError := (nErrorId <> BACnet_ERR_NO_ERROR);

END_FUNCTION_BLOCK

// POUs/BACnet Objects/Remote (Client)/Extended Process Data/FB_BACnet_RemoteGroup_EX
FUNCTION_BLOCK FB_BACnet_RemoteGroup_EX
VAR_IN_OUT
	RemoteDevice		: FB_BACnet_RemoteDevice;
END_VAR
VAR_OUTPUT
	bReady				: BOOL;
	tObjectID			: T_BACnet_ObjectIdentifier := 16#FFFFFFFF;
	bError				: BOOL;
	nErrorId			: UINT;
END_VAR
VAR
	_ObjectId AT%I*: DWORD;			(* ~(BACnet_ObjectIdentifier:		: LINK)
										(BACNET_OBJECTTYPE		: GROUP : ) *)
	_nUpdateCount : UDINT := 0;
END_VAR

(* update client device *)
IF RemoteDevice._nUpdateCount = _nUpdateCount THEN
	RemoteDevice();
END_IF
(* remind current number of update counter *)
_nUpdateCount := RemoteDevice._nUpdateCount;

IF NOT RemoteDevice.bOperational THEN
	(* server device not ready, reset local ready also *)
	bReady := FALSE;
	(* and set error ID *)
	nErrorId := BACnet_ERR_OPERATIONAL;

